LIN {X 0,Y 232.214,Z 369.64,A -85,B 0,C 180,E1 -19869.961,E2 -19869.961} C_VEL
LIN {X 0,Y 230.264,Z 376.571,A -85,B 0,C 180,E1 -19872.229,E2 -19872.229} C_VEL
LIN {X 0,Y 229.077,Z 381.074,A -85,B 0,C 180,E1 -19873.972,E2 -19873.972} C_VEL
LIN {X 0,Y 227.545,Z 386.565,A -85,B 0,C 180,E1 -19876.606,E2 -19876.606} C_VEL
LIN {X 0,Y 226.573,Z 390.894,A -85,B 0,C 180,E1 -19879.274,E2 -19879.274} C_VEL
LIN {X 0,Y 226.135,Z 393.264,A -85,B 0,C 180,E1 -19881.06,E2 -19881.06} C_VEL
LIN {X 0,Y 225.811,Z 395.066,A -85,B 0,C 180,E1 -19882.849,E2 -19882.849} C_VEL
LIN {X 0,Y 225.588,Z 397.52,A -85,B 0,C 180,E1 -19886.428,E2 -19886.428} C_VEL
LIN {X 0,Y 225.625,Z 398.113,A -85,B 0,C 180,E1 -19888.215,E2 -19888.215} C_VEL
LIN {X 0,Y 225.708,Z 398.27,A -85,B 0,C 180,E1 -19890,E2 -19890} C_VEL
LIN {X 0,Y 225.624,Z 398.113,A -85,B 0,C 180,E1 -19891.785,E2 -19891.785} C_VEL
LIN {X 0,Y 225.587,Z 397.046,A -85,B 0,C 180,E1 -19894.475,E2 -19894.475} C_VEL
LIN {X 0,Y 225.778,Z 395.065,A -85,B 0,C 180,E1 -19897.152,E2 -19897.152} C_VEL
LIN {X 0,Y 226.327,Z 392.112,A -85,B 0,C 180,E1 -19899.834,E2 -19899.834} C_VEL
LIN {X 0,Y 227.177,Z 388.12,A -85,B 0,C 180,E1 -19902.507,E2 -19902.507} C_VEL
LIN {X 0,Y 228.512,Z 382.989,A -85,B 0,C 180,E1 -19905.154,E2 -19905.154} C_VEL
LIN {X 0,Y 229.992,Z 377.728,A -85,B 0,C 180,E1 -19907.334,E2 -19907.334} C_VEL
LIN {X 0,Y 231.748,Z 371.413,A -85,B 0,C 180,E1 -19909.486,E2 -19909.486} C_VEL
LIN {X 0,Y 233.277,Z 365.461,A -85,B 0,C 180,E1 -19911.194,E2 -19911.194} C_VEL
LIN {X 0,Y 235.024,Z 358.534,A -85,B 0,C 180,E1 -19912.876,E2 -19912.876} C_VEL
LIN {X 0,Y 237.101,Z 350.359,A -85,B 0,C 180,E1 -19914.518,E2 -19914.518} C_VEL
LIN {X 0,Y 239.016,Z 341.85,A -85,B 0,C 180,E1 -19915.937,E2 -19915.937} C_VEL
LIN {X 0,Y 240.893,Z 333.14,A -85,B 0,C 180,E1 -19917.12,E2 -19917.12} C_VEL
LIN {X 0,Y 242.62,Z 323.384,A -85,B 0,C 180,E1 -19918.198,E2 -19918.198} C_VEL
LIN {X 0,Y 244.14,Z 313.306,A -85,B 0,C 180,E1 -19919.063,E2 -19919.063} C_VEL
LIN {X 0,Y 245.33,Z 303.86,A -85,B 0,C 180,E1 -19919.669,E2 -19919.669} C_VEL
LIN {X 0,Y 246.133,Z 293.823,A -85,B 0,C 180,E1 -19920.141,E2 -19920.141} C_VEL
LIN {X 0,Y 247.891,Z 250.011,A -85,B 0,C 180,E1 -19921.412,E2 -19921.412} C_VEL
LIN {X 0,Y 248.127,Z 242.633,A -85,B 0,C 180,E1 -19921.624,E2 -19921.624} C_VEL
LIN {X 0,Y 244.357,Z 220.685,A -85,B 0,C 180,E1 -19922.914,E2 -19922.914} C_VEL
LIN {X 0,Y 243.134,Z 215.724,A -85,B 0,C 180,E1 -19923.271,E2 -19923.271} C_VEL
LIN {X 0,Y 235.991,Z 199.45,A -85,B 0,C 180,E1 -19924.997,E2 -19924.997} C_VEL
LIN {X 0,Y 230.184,Z 187.454,A -85,B 0,C 180,E1 -19926.503,E2 -19926.503} C_VEL
LIN {X 0,Y 229.739,Z 185.681,A -85,B 0,C 180,E1 -19927.308,E2 -19927.308} C_VEL
LIN {X 0,Y 228.311,Z 179.722,A -85,B 0,C 180,E1 -19931.046,E2 -19931.046} C_VEL
LIN {X 0,Y 227.848,Z 177.605,A -85,B 0,C 180,E1 -19932.574,E2 -19932.574} C_VEL
LIN {X 0,Y 227.808,Z 177.611,A -85,B 0,C 180,E1 -19937.256,E2 -19937.256} C_VEL
LIN {X 0,Y 227.846,Z 177.6,A -85,B 0,C 180,E1 -19941.908,E2 -19941.908} C_VEL
LIN {X 0,Y 227.881,Z 177.572,A -85,B 0,C 180,E1 -19946.376,E2 -19946.376} C_VEL
LIN {X 0,Y 227.918,Z 177.586,A -85,B 0,C 180,E1 -19950.437,E2 -19950.437} C_VEL
LIN {X 0,Y 227.929,Z 177.566,A -85,B 0,C 180,E1 -19954.425,E2 -19954.425} C_VEL
LIN {X 0,Y 227.962,Z 177.578,A -85,B 0,C 180,E1 -19958.286,E2 -19958.286} C_VEL
LIN {X 0,Y 228.034,Z 177.546,A -85,B 0,C 180,E1 -19962.825,E2 -19962.825} C_VEL
LIN {X 0,Y 228.072,Z 177.558,A -85,B 0,C 180,E1 -19967.542,E2 -19967.542} C_VEL
LIN {X 0,Y 228.266,Z 177.506,A -85,B 0,C 180,E1 -19971.144,E2 -19971.144} C_VEL
LIN {X 0,Y 228.323,Z 177.524,A -85,B 0,C 180,E1 -19972.927,E2 -19972.927} C_VEL
LIN {X 0,Y 228.552,Z 177.483,A -85,B 0,C 180,E1 -19978.237,E2 -19978.237} C_VEL
LIN {X 0,Y 228.553,Z 177.478,A -85,B 0,C 180,E1 -19981.761,E2 -19981.761} C_VEL
LIN {X 0,Y 228.353,Z 177.524,A -85,B 0,C 180,E1 -19987.07,E2 -19987.07} C_VEL
LIN {X 0,Y 228.161,Z 177.521,A -85,B 0,C 180,E1 -19990.649,E2 -19990.649} C_VEL
LIN {X 0,Y 228.062,Z 177.578,A -85,B 0,C 180,E1 -19994.271,E2 -19994.271} C_VEL
LIN {X 0,Y 228,Z 177.547,A -85,B 0,C 180,E1 -19997.952,E2 -19997.952} C_VEL
LIN {X 0,Y 227.927,Z 177.588,A -85,B 0,C 180,E1 -20002.329,E2 -20002.329} C_VEL
LIN {X 0,Y 227.94,Z 177.56,A -85,B 0,C 180,E1 -20006.602,E2 -20006.602} C_VEL
LIN {X 0,Y 227.906,Z 177.594,A -85,B 0,C 180,E1 -20010.295,E2 -20010.295} C_VEL
LIN {X 0,Y 227.886,Z 177.573,A -85,B 0,C 180,E1 -20013.718,E2 -20013.718} C_VEL
LIN {X 0,Y 227.866,Z 177.602,A -85,B 0,C 180,E1 -20018.085,E2 -20018.085} C_VEL
LIN {X 0,Y 227.812,Z 177.605,A -85,B 0,C 180,E1 -20022.741,E2 -20022.741} C_VEL
LIN {X 0,Y 227.811,Z 177.543,A -85,B 0,C 180,E1 -20027.258,E2 -20027.258} C_VEL
LIN {X 0,Y 227.866,Z 177.603,A -85,B 0,C 180,E1 -20031.914,E2 -20031.914} C_VEL
LIN {X 0,Y 227.929,Z 177.929,A -85,B 0,C 180,E1 -20032.938,E2 -20032.938} C_VEL
LIN {X 0,Y 228.316,Z 179.228,A -85,B 0,C 180,E1 -20033.246,E2 -20033.246} C_VEL
LIN {X 0,Y 230.062,Z 181.874,A -85,B 0,C 180,E1 -20033.684,E2 -20033.684} C_VEL
LIN {X 0,Y 239.018,Z 197.391,A -85,B 0,C 180,E1 -20035.813,E2 -20035.813} C_VEL
LIN {X 0,Y 245.285,Z 209.395,A -85,B 0,C 180,E1 -20037.22,E2 -20037.22} C_VEL
LIN {X 0,Y 252.548,Z 222.93,A -85,B 0,C 180,E1 -20038.725,E2 -20038.725} C_VEL
LIN {X 0,Y 261.317,Z 235.879,A -85,B 0,C 180,E1 -20040.298,E2 -20040.298} C_VEL
LIN {X 0,Y 272.635,Z 249.159,A -85,B 0,C 180,E1 -20042.045,E2 -20042.045} C_VEL
LIN {X 0,Y 286.641,Z 263.214,A -85,B 0,C 180,E1 -20043.918,E2 -20043.918} C_VEL
LIN {X 0,Y 299.817,Z 274.419,A -85,B 0,C 180,E1 -20045.476,E2 -20045.476} C_VEL
LIN {X 0,Y 307.547,Z 280.739,A -85,B 0,C 180,E1 -20046.479,E2 -20046.479} C_VEL
LIN {X 0,Y 315.797,Z 287.099,A -85,B 0,C 180,E1 -20047.77,E2 -20047.77} C_VEL
LIN {X 0,Y 323.581,Z 292.925,A -85,B 0,C 180,E1 -20049.173,E2 -20049.173} C_VEL
LIN {X 0,Y 331.85,Z 299.062,A -85,B 0,C 180,E1 -20050.874,E2 -20050.874} C_VEL
LIN {X 0,Y 339.226,Z 304.074,A -85,B 0,C 180,E1 -20052.563,E2 -20052.563} C_VEL
LIN {X 0,Y 345.901,Z 309.055,A -85,B 0,C 180,E1 -20054.348,E2 -20054.348} C_VEL
LIN {X 0,Y 351.923,Z 312.847,A -85,B 0,C 180,E1 -20056.135,E2 -20056.135} C_VEL
LIN {X 0,Y 355.943,Z 315.097,A -85,B 0,C 180,E1 -20057.456,E2 -20057.456} C_VEL
LIN {X 0,Y 359.121,Z 317.594,A -85,B 0,C 180,E1 -20058.715,E2 -20058.715} C_VEL
LIN {X 0,Y 363.313,Z 320.464,A -85,B 0,C 180,E1 -20060.589,E2 -20060.589} C_VEL
LIN {X 0,Y 366.561,Z 322.302,A -85,B 0,C 180,E1 -20062.287,E2 -20062.287} C_VEL
LIN {X 0,Y 368.408,Z 323.209,A -85,B 0,C 180,E1 -20063.428,E2 -20063.428} C_VEL
LIN {X 0,Y 369.964,Z 323.883,A -85,B 0,C 180,E1 -20064.55,E2 -20064.55} C_VEL
LIN {X 0,Y 371.235,Z 324.349,A -85,B 0,C 180,E1 -20065.657,E2 -20065.657} C_VEL
LIN {X 0,Y 372.231,Z 324.627,A -85,B 0,C 180,E1 -20066.753,E2 -20066.753} C_VEL
LIN {X 0,Y 372.866,Z 324.996,A -85,B 0,C 180,E1 -20067.84,E2 -20067.84} C_VEL
LIN {X 0,Y 373.221,Z 325.279,A -85,B 0,C 180,E1 -20068.921,E2 -20068.921} C_VEL
LIN {X 0,Y 373.406,Z 325.182,A -85,B 0,C 180,E1 -20070,E2 -20070} C_VEL
LIN {X 0,Y 373.242,Z 325.214,A -85,B 0,C 180,E1 -20071.079,E2 -20071.079} C_VEL
LIN {X 0,Y 372.792,Z 324.929,A -85,B 0,C 180,E1 -20072.349,E2 -20072.349} C_VEL
LIN {X 0,Y 371.247,Z 324.325,A -85,B 0,C 180,E1 -20074.343,E2 -20074.343} C_VEL
LIN {X 0,Y 369.974,Z 323.88,A -85,B 0,C 180,E1 -20075.45,E2 -20075.45} C_VEL
LIN {X 0,Y 368.057,Z 323.044,A -85,B 0,C 180,E1 -20076.821,E2 -20076.821} C_VEL
LIN {X 0,Y 366.574,Z 322.333,A -85,B 0,C 180,E1 -20077.713,E2 -20077.713} C_VEL
LIN {X 0,Y 363.308,Z 320.439,A -85,B 0,C 180,E1 -20079.406,E2 -20079.406} C_VEL
LIN {X 0,Y 359.112,Z 317.577,A -85,B 0,C 180,E1 -20081.286,E2 -20081.286} C_VEL
LIN {X 0,Y 355.896,Z 315.079,A -85,B 0,C 180,E1 -20082.546,E2 -20082.546} C_VEL
LIN {X 0,Y 351.917,Z 312.837,A -85,B 0,C 180,E1 -20083.866,E2 -20083.866} C_VEL
LIN {X 0,Y 345.745,Z 308.908,A -85,B 0,C 180,E1 -20085.699,E2 -20085.699} C_VEL
LIN {X 0,Y 338.798,Z 303.827,A -85,B 0,C 180,E1 -20087.534,E2 -20087.534} C_VEL
LIN {X 0,Y 330.886,Z 298.432,A -85,B 0,C 180,E1 -20089.33,E2 -20089.33} C_VEL
LIN {X 0,Y 323.177,Z 292.616,A -85,B 0,C 180,E1 -20090.901,E2 -20090.901} C_VEL
LIN {X 0,Y 315.363,Z 286.776,A -85,B 0,C 180,E1 -20092.3,E2 -20092.3} C_VEL
LIN {X 0,Y 306.83,Z 280.18,A -85,B 0,C 180,E1 -20093.624,E2 -20093.624} C_VEL
LIN {X 0,Y 298.134,Z 273.077,A -85,B 0,C 180,E1 -20094.73,E2 -20094.73} C_VEL
LIN {X 0,Y 282.857,Z 259.613,A -85,B 0,C 180,E1 -20096.561,E2 -20096.561} C_VEL
LIN {X 0,Y 269.247,Z 245.479,A -85,B 0,C 180,E1 -20098.451,E2 -20098.451} C_VEL
LIN {X 0,Y 260.422,Z 234.592,A -85,B 0,C 180,E1 -20099.856,E2 -20099.856} C_VEL
LIN {X 0,Y 252.398,Z 222.675,A -85,B 0,C 180,E1 -20101.304,E2 -20101.304} C_VEL
LIN {X 0,Y 245.458,Z 209.83,A -85,B 0,C 180,E1 -20102.739,E2 -20102.739} C_VEL
LIN {X 0,Y 239.261,Z 197.815,A -85,B 0,C 180,E1 -20104.132,E2 -20104.132} C_VEL
LIN {X 0,Y 231.588,Z 184.592,A -85,B 0,C 180,E1 -20105.935,E2 -20105.935} C_VEL
LIN {X 0,Y 229.701,Z 181.488,A -85,B 0,C 180,E1 -20106.397,E2 -20106.397} C_VEL
LIN {X 0,Y 228.091,Z 178.529,A -85,B 0,C 180,E1 -20106.86,E2 -20106.86} C_VEL
LIN {X 0,Y 227.9,Z 177.655,A -85,B 0,C 180,E1 -20107.312,E2 -20107.312} C_VEL
LIN {X 0,Y 227.829,Z 177.552,A -85,B 0,C 180,E1 -20110.375,E2 -20110.375} C_VEL
LIN {X 0,Y 227.832,Z 177.581,A -85,B 0,C 180,E1 -20115.193,E2 -20115.193} C_VEL
LIN {X 0,Y 227.83,Z 177.584,A -85,B 0,C 180,E1 -20119.625,E2 -20119.625} C_VEL
LIN {X 0,Y 227.896,Z 177.578,A -85,B 0,C 180,E1 -20124.132,E2 -20124.132} C_VEL
LIN {X 0,Y 227.87,Z 177.6,A -85,B 0,C 180,E1 -20128.379,E2 -20128.379} C_VEL
LIN {X 0,Y 227.883,Z 177.565,A -85,B 0,C 180,E1 -20132.446,E2 -20132.446} C_VEL
LIN {X 0,Y 227.911,Z 177.596,A -85,B 0,C 180,E1 -20136.368,E2 -20136.368} C_VEL
LIN {X 0,Y 227.939,Z 177.552,A -85,B 0,C 180,E1 -20140.175,E2 -20140.175} C_VEL
LIN {X 0,Y 228.055,Z 177.569,A -85,B 0,C 180,E1 -20143.899,E2 -20143.899} C_VEL
LIN {X 0,Y 228.092,Z 177.554,A -85,B 0,C 180,E1 -20147.545,E2 -20147.545} C_VEL
LIN {X 0,Y 228.304,Z 177.505,A -85,B 0,C 180,E1 -20151.147,E2 -20151.147} C_VEL
LIN {X 0,Y 228.353,Z 177.524,A -85,B 0,C 180,E1 -20152.93,E2 -20152.93} C_VEL
LIN {X 0,Y 228.553,Z 177.478,A -85,B 0,C 180,E1 -20158.239,E2 -20158.239} C_VEL
LIN {X 0,Y 228.552,Z 177.483,A -85,B 0,C 180,E1 -20161.763,E2 -20161.763} C_VEL
LIN {X 0,Y 228.323,Z 177.524,A -85,B 0,C 180,E1 -20167.073,E2 -20167.073} C_VEL
LIN {X 0,Y 228.145,Z 177.523,A -85,B 0,C 180,E1 -20170.652,E2 -20170.652} C_VEL
LIN {X 0,Y 228.064,Z 177.573,A -85,B 0,C 180,E1 -20174.273,E2 -20174.273} C_VEL
LIN {X 0,Y 228.003,Z 177.542,A -85,B 0,C 180,E1 -20177.954,E2 -20177.954} C_VEL
LIN {X 0,Y 227.93,Z 177.589,A -85,B 0,C 180,E1 -20182.33,E2 -20182.33} C_VEL
LIN {X 0,Y 227.943,Z 177.556,A -85,B 0,C 180,E1 -20186.604,E2 -20186.604} C_VEL
LIN {X 0,Y 227.908,Z 177.595,A -85,B 0,C 180,E1 -20190.297,E2 -20190.297} C_VEL
LIN {X 0,Y 227.879,Z 177.572,A -85,B 0,C 180,E1 -20193.721,E2 -20193.721} C_VEL
LIN {X 0,Y 227.846,Z 177.6,A -85,B 0,C 180,E1 -20198.092,E2 -20198.092} C_VEL
LIN {X 0,Y 227.808,Z 177.609,A -85,B 0,C 180,E1 -20202.744,E2 -20202.744} C_VEL
LIN {X 0,Y 227.85,Z 177.623,A -85,B 0,C 180,E1 -20207.506,E2 -20207.506} C_VEL
LIN {X 0,Y 229.254,Z 183.3,A -85,B 0,C 180,E1 -20211.23,E2 -20211.23} C_VEL
LIN {X 0,Y 230.082,Z 187.069,A -85,B 0,C 180,E1 -20213.403,E2 -20213.403} C_VEL
LIN {X 0,Y 231.752,Z 190.832,A -85,B 0,C 180,E1 -20213.949,E2 -20213.949} C_VEL
LIN {X 0,Y 238.601,Z 205.182,A -85,B 0,C 180,E1 -20215.643,E2 -20215.643} C_VEL
LIN {X 0,Y 243.547,Z 216.733,A -85,B 0,C 180,E1 -20216.827,E2 -20216.827} C_VEL
LIN {X 0,Y 247.169,Z 236.517,A -85,B 0,C 180,E1 -20218.035,E2 -20218.035} C_VEL
LIN {X 0,Y 248.164,Z 243.57,A -85,B 0,C 180,E1 -20218.412,E2 -20218.412} C_VEL
LIN {X 0,Y 248.06,Z 246.228,A -85,B 0,C 180,E1 -20218.486,E2 -20218.486} C_VEL
LIN {X 0,Y 247.255,Z 252.073,A -85,B 0,C 180,E1 -20218.567,E2 -20218.567} C_VEL
LIN {X 0,Y 241.602,Z 271.074,A -85,B 0,C 180,E1 -20218.4,E2 -20218.4} C_VEL
LIN {X 0,Y 240.823,Z 276.917,A -85,B 0,C 180,E1 -20218.487,E2 -20218.487} C_VEL
LIN {X 0,Y 239.896,Z 296.606,A -85,B 0,C 180,E1 -20219.126,E2 -20219.126} C_VEL
LIN {X 0,Y 238.338,Z 310.54,A -85,B 0,C 180,E1 -20219.915,E2 -20219.915} C_VEL
LIN {X 0,Y 236.759,Z 321.18,A -85,B 0,C 180,E1 -20220.795,E2 -20220.795} C_VEL
LIN {X 0,Y 235.242,Z 329.685,A -85,B 0,C 180,E1 -20221.688,E2 -20221.688} C_VEL
LIN {X 0,Y 233.324,Z 338.958,A -85,B 0,C 180,E1 -20222.898,E2 -20222.898} C_VEL
LIN {X 0,Y 231.165,Z 347.897,A -85,B 0,C 180,E1 -20224.327,E2 -20224.327} C_VEL
LIN {X 0,Y 228.986,Z 356.423,A -85,B 0,C 180,E1 -20226.005,E2 -20226.005} C_VEL
LIN {X 0,Y 227.032,Z 363.64,A -85,B 0,C 180,E1 -20227.715,E2 -20227.715} C_VEL
LIN {X 0,Y 225.349,Z 370.062,A -85,B 0,C 180,E1 -20229.536,E2 -20229.536} C_VEL
LIN {X 0,Y 223.482,Z 376.379,A -85,B 0,C 180,E1 -20231.671,E2 -20231.671} C_VEL
LIN {X 0,Y 222.246,Z 380.882,A -85,B 0,C 180,E1 -20233.465,E2 -20233.465} C_VEL
LIN {X 0,Y 220.607,Z 386.372,A -85,B 0,C 180,E1 -20236.177,E2 -20236.177} C_VEL
LIN {X 0,Y 219.584,Z 390.702,A -85,B 0,C 180,E1 -20238.929,E2 -20238.929} C_VEL
LIN {X 0,Y 219.086,Z 393.072,A -85,B 0,C 180,E1 -20240.77,E2 -20240.77} C_VEL
LIN {X 0,Y 218.737,Z 394.874,A -85,B 0,C 180,E1 -20242.616,E2 -20242.616} C_VEL
LIN {X 0,Y 218.501,Z 397.328,A -85,B 0,C 180,E1 -20246.312,E2 -20246.312} C_VEL
LIN {X 0,Y 218.525,Z 397.921,A -85,B 0,C 180,E1 -20248.157,E2 -20248.157} C_VEL
LIN {X 0,Y 218.623,Z 398.079,A -85,B 0,C 180,E1 -20250,E2 -20250} C_VEL
LIN {X 0,Y 218.524,Z 397.921,A -85,B 0,C 180,E1 -20251.843,E2 -20251.843} C_VEL
LIN {X 0,Y 218.484,Z 397.064,A -85,B 0,C 180,E1 -20254.292,E2 -20254.292} C_VEL
LIN {X 0,Y 218.705,Z 394.873,A -85,B 0,C 180,E1 -20257.385,E2 -20257.385} C_VEL
LIN {X 0,Y 219.313,Z 391.92,A -85,B 0,C 180,E1 -20260.151,E2 -20260.151} C_VEL
LIN {X 0,Y 220.202,Z 387.927,A -85,B 0,C 180,E1 -20262.909,E2 -20262.909} C_VEL
LIN {X 0,Y 221.652,Z 382.797,A -85,B 0,C 180,E1 -20265.635,E2 -20265.635} C_VEL
LIN {X 0,Y 223.161,Z 377.535,A -85,B 0,C 180,E1 -20267.882,E2 -20267.882} C_VEL
LIN {X 0,Y 225.05,Z 371.221,A -85,B 0,C 180,E1 -20270.091,E2 -20270.091} C_VEL
LIN {X 0,Y 226.622,Z 365.268,A -85,B 0,C 180,E1 -20271.848,E2 -20271.848} C_VEL
LIN {X 0,Y 228.474,Z 358.341,A -85,B 0,C 180,E1 -20273.571,E2 -20273.571} C_VEL
LIN {X 0,Y 230.662,Z 350.168,A -85,B 0,C 180,E1 -20275.249,E2 -20275.249} C_VEL
LIN {X 0,Y 232.638,Z 341.658,A -85,B 0,C 180,E1 -20276.703,E2 -20276.703} C_VEL
LIN {X 0,Y 234.602,Z 332.948,A -85,B 0,C 180,E1 -20277.909,E2 -20277.909} C_VEL
LIN {X 0,Y 236.379,Z 323.192,A -85,B 0,C 180,E1 -20279.012,E2 -20279.012} C_VEL
LIN {X 0,Y 237.942,Z 313.114,A -85,B 0,C 180,E1 -20279.896,E2 -20279.896} C_VEL
LIN {X 0,Y 239.227,Z 303.118,A -85,B 0,C 180,E1 -20280.544,E2 -20280.544} C_VEL
LIN {X 0,Y 240.04,Z 293.142,A -85,B 0,C 180,E1 -20281.012,E2 -20281.012} C_VEL
LIN {X 0,Y 242.113,Z 243.843,A -85,B 0,C 180,E1 -20282.457,E2 -20282.457} C_VEL
LIN {X 0,Y 238.247,Z 221.322,A -85,B 0,C 180,E1 -20283.841,E2 -20283.841} C_VEL
LIN {X 0,Y 237.362,Z 218.29,A -85,B 0,C 180,E1 -20284.091,E2 -20284.091} C_VEL
LIN {X 0,Y 230.872,Z 203.304,A -85,B 0,C 180,E1 -20285.74,E2 -20285.74} C_VEL
LIN {X 0,Y 224.409,Z 190.406,A -85,B 0,C 180,E1 -20287.434,E2 -20287.434} C_VEL
LIN {X 0,Y 222.782,Z 186.821,A -85,B 0,C 180,E1 -20288.007,E2 -20288.007} C_VEL
LIN {X 0,Y 221.299,Z 180.788,A -85,B 0,C 180,E1 -20291.829,E2 -20291.829} C_VEL
LIN {X 0,Y 220.782,Z 178.503,A -85,B 0,C 180,E1 -20293.481,E2 -20293.481} C_VEL
LIN {X 0,Y 220.768,Z 178.482,A -85,B 0,C 180,E1 -20298.046,E2 -20298.046} C_VEL
LIN {X 0,Y 220.825,Z 178.479,A -85,B 0,C 180,E1 -20302.792,E2 -20302.792} C_VEL
LIN {X 0,Y 220.819,Z 178.459,A -85,B 0,C 180,E1 -20307.243,E2 -20307.243} C_VEL
LIN {X 0,Y 220.836,Z 178.451,A -85,B 0,C 180,E1 -20311.485,E2 -20311.485} C_VEL
LIN {X 0,Y 220.868,Z 178.46,A -85,B 0,C 180,E1 -20315.564,E2 -20315.564} C_VEL
LIN {X 0,Y 220.892,Z 178.438,A -85,B 0,C 180,E1 -20319.513,E2 -20319.513} C_VEL
LIN {X 0,Y 221.016,Z 178.427,A -85,B 0,C 180,E1 -20323.369,E2 -20323.369} C_VEL
LIN {X 0,Y 221.011,Z 178.444,A -85,B 0,C 180,E1 -20327.138,E2 -20327.138} C_VEL
LIN {X 0,Y 221.204,Z 178.383,A -85,B 0,C 180,E1 -20330.858,E2 -20330.858} C_VEL
LIN {X 0,Y 221.258,Z 178.398,A -85,B 0,C 180,E1 -20332.7,E2 -20332.7} C_VEL
LIN {X 0,Y 221.51,Z 178.36,A -85,B 0,C 180,E1 -20338.181,E2 -20338.181} C_VEL
LIN {X 0,Y 221.511,Z 178.355,A -85,B 0,C 180,E1 -20341.817,E2 -20341.817} C_VEL
LIN {X 0,Y 221.288,Z 178.399,A -85,B 0,C 180,E1 -20347.297,E2 -20347.297} C_VEL
LIN {X 0,Y 221.11,Z 178.401,A -85,B 0,C 180,E1 -20350.993,E2 -20350.993} C_VEL
LIN {X 0,Y 221.014,Z 178.436,A -85,B 0,C 180,E1 -20356.629,E2 -20356.629} C_VEL
LIN {X 0,Y 220.89,Z 178.436,A -85,B 0,C 180,E1 -20360.485,E2 -20360.485} C_VEL
LIN {X 0,Y 220.865,Z 178.469,A -85,B 0,C 180,E1 -20364.434,E2 -20364.434} C_VEL
LIN {X 0,Y 220.833,Z 178.449,A -85,B 0,C 180,E1 -20368.513,E2 -20368.513} C_VEL
LIN {X 0,Y 220.821,Z 178.463,A -85,B 0,C 180,E1 -20372.754,E2 -20372.754} C_VEL
LIN {X 0,Y 220.835,Z 178.477,A -85,B 0,C 180,E1 -20377.287,E2 -20377.287} C_VEL
LIN {X 0,Y 220.772,Z 178.47,A -85,B 0,C 180,E1 -20381.951,E2 -20381.951} C_VEL
LIN {X 0,Y 220.772,Z 178.441,A -85,B 0,C 180,E1 -20385.546,E2 -20385.546} C_VEL
LIN {X 0,Y 220.805,Z 178.44,A -85,B 0,C 180,E1 -20390.463,E2 -20390.463} C_VEL
LIN {X 0,Y 220.869,Z 178.776,A -85,B 0,C 180,E1 -20391.555,E2 -20391.555} C_VEL
LIN {X 0,Y 221.231,Z 180.131,A -85,B 0,C 180,E1 -20391.89,E2 -20391.89} C_VEL
LIN {X 0,Y 222.982,Z 182.764,A -85,B 0,C 180,E1 -20392.361,E2 -20392.361} C_VEL
LIN {X 0,Y 230.22,Z 194.713,A -85,B 0,C 180,E1 -20394.2,E2 -20394.2} C_VEL
LIN {X 0,Y 238.43,Z 209.905,A -85,B 0,C 180,E1 -20396.163,E2 -20396.163} C_VEL
LIN {X 0,Y 246.332,Z 225.31,A -85,B 0,C 180,E1 -20397.917,E2 -20397.917} C_VEL
LIN {X 0,Y 254.125,Z 237.265,A -85,B 0,C 180,E1 -20399.406,E2 -20399.406} C_VEL
LIN {X 0,Y 261.098,Z 246.325,A -85,B 0,C 180,E1 -20400.594,E2 -20400.594} C_VEL
LIN {X 0,Y 272.34,Z 258.902,A -85,B 0,C 180,E1 -20402.297,E2 -20402.297} C_VEL
LIN {X 0,Y 285.178,Z 271.16,A -85,B 0,C 180,E1 -20403.991,E2 -20403.991} C_VEL
LIN {X 0,Y 298.365,Z 282.288,A -85,B 0,C 180,E1 -20405.579,E2 -20405.579} C_VEL
LIN {X 0,Y 306.925,Z 289.092,A -85,B 0,C 180,E1 -20406.771,E2 -20406.771} C_VEL
LIN {X 0,Y 315.592,Z 295.809,A -85,B 0,C 180,E1 -20408.207,E2 -20408.207} C_VEL
LIN {X 0,Y 323.961,Z 301.874,A -85,B 0,C 180,E1 -20409.783,E2 -20409.783} C_VEL
LIN {X 0,Y 331.81,Z 307.611,A -85,B 0,C 180,E1 -20411.476,E2 -20411.476} C_VEL
LIN {X 0,Y 338.558,Z 312.236,A -85,B 0,C 180,E1 -20413.105,E2 -20413.105} C_VEL
LIN {X 0,Y 343.959,Z 316.177,A -85,B 0,C 180,E1 -20414.596,E2 -20414.596} C_VEL
LIN {X 0,Y 348.699,Z 319.119,A -85,B 0,C 180,E1 -20416.004,E2 -20416.004} C_VEL
LIN {X 0,Y 352.904,Z 321.471,A -85,B 0,C 180,E1 -20417.372,E2 -20417.372} C_VEL
LIN {X 0,Y 357.621,Z 325.06,A -85,B 0,C 180,E1 -20419.293,E2 -20419.293} C_VEL
LIN {X 0,Y 361.369,Z 327.489,A -85,B 0,C 180,E1 -20421.049,E2 -20421.049} C_VEL
LIN {X 0,Y 363.545,Z 328.713,A -85,B 0,C 180,E1 -20422.223,E2 -20422.223} C_VEL
LIN {X 0,Y 365.441,Z 329.628,A -85,B 0,C 180,E1 -20423.374,E2 -20423.374} C_VEL
LIN {X 0,Y 367.1,Z 330.364,A -85,B 0,C 180,E1 -20424.568,E2 -20424.568} C_VEL
LIN {X 0,Y 368.306,Z 330.811,A -85,B 0,C 180,E1 -20425.623,E2 -20425.623} C_VEL
LIN {X 0,Y 369.322,Z 331.105,A -85,B 0,C 180,E1 -20426.727,E2 -20426.727} C_VEL
LIN {X 0,Y 369.972,Z 331.455,A -85,B 0,C 180,E1 -20427.823,E2 -20427.823} C_VEL
LIN {X 0,Y 370.325,Z 331.734,A -85,B 0,C 180,E1 -20428.913,E2 -20428.913} C_VEL
LIN {X 0,Y 370.523,Z 331.644,A -85,B 0,C 180,E1 -20430,E2 -20430} C_VEL
LIN {X 0,Y 370.339,Z 331.689,A -85,B 0,C 180,E1 -20431.087,E2 -20431.087} C_VEL
LIN {X 0,Y 369.977,Z 331.421,A -85,B 0,C 180,E1 -20432.177,E2 -20432.177} C_VEL
LIN {X 0,Y 369.32,Z 331.082,A -85,B 0,C 180,E1 -20433.273,E2 -20433.273} C_VEL
LIN {X 0,Y 368.309,Z 330.779,A -85,B 0,C 180,E1 -20434.377,E2 -20434.377} C_VEL
LIN {X 0,Y 367.016,Z 330.323,A -85,B 0,C 180,E1 -20435.494,E2 -20435.494} C_VEL
LIN {X 0,Y 365.437,Z 329.642,A -85,B 0,C 180,E1 -20436.626,E2 -20436.626} C_VEL
LIN {X 0,Y 362.342,Z 328.045,A -85,B 0,C 180,E1 -20438.435,E2 -20438.435} C_VEL
LIN {X 0,Y 358.864,Z 325.916,A -85,B 0,C 180,E1 -20440.152,E2 -20440.152} C_VEL
LIN {X 0,Y 354.955,Z 323.141,A -85,B 0,C 180,E1 -20441.812,E2 -20441.812} C_VEL
LIN {X 0,Y 352.801,Z 321.444,A -85,B 0,C 180,E1 -20442.658,E2 -20442.658} C_VEL
LIN {X 0,Y 347.992,Z 318.709,A -85,B 0,C 180,E1 -20444.213,E2 -20444.213} C_VEL
LIN {X 0,Y 343.044,Z 315.551,A -85,B 0,C 180,E1 -20445.66,E2 -20445.66} C_VEL
LIN {X 0,Y 338.086,Z 311.947,A -85,B 0,C 180,E1 -20447.017,E2 -20447.017} C_VEL
LIN {X 0,Y 330.772,Z 306.921,A -85,B 0,C 180,E1 -20448.753,E2 -20448.753} C_VEL
LIN {X 0,Y 323.263,Z 301.326,A -85,B 0,C 180,E1 -20450.356,E2 -20450.356} C_VEL
LIN {X 0,Y 314.609,Z 295.066,A -85,B 0,C 180,E1 -20451.969,E2 -20451.969} C_VEL
LIN {X 0,Y 306.168,Z 288.54,A -85,B 0,C 180,E1 -20453.34,E2 -20453.34} C_VEL
LIN {X 0,Y 298.371,Z 282.29,A -85,B 0,C 180,E1 -20454.423,E2 -20454.423} C_VEL
LIN {X 0,Y 286.498,Z 272.292,A -85,B 0,C 180,E1 -20455.848,E2 -20455.848} C_VEL
LIN {X 0,Y 276.553,Z 263.037,A -85,B 0,C 180,E1 -20457.124,E2 -20457.124} C_VEL
LIN {X 0,Y 264.555,Z 250.461,A -85,B 0,C 180,E1 -20458.856,E2 -20458.856} C_VEL
LIN {X 0,Y 255.684,Z 239.447,A -85,B 0,C 180,E1 -20460.317,E2 -20460.317} C_VEL
LIN {X 0,Y 247.844,Z 227.763,A -85,B 0,C 180,E1 -20461.781,E2 -20461.781} C_VEL
LIN {X 0,Y 241.06,Z 215.332,A -85,B 0,C 180,E1 -20463.226,E2 -20463.226} C_VEL
LIN {X 0,Y 234.477,Z 202.332,A -85,B 0,C 180,E1 -20464.769,E2 -20464.769} C_VEL
LIN {X 0,Y 225.477,Z 186.693,A -85,B 0,C 180,E1 -20466.994,E2 -20466.994} C_VEL
LIN {X 0,Y 222.661,Z 182.415,A -85,B 0,C 180,E1 -20467.717,E2 -20467.717} C_VEL
LIN {X 0,Y 221.064,Z 179.607,A -85,B 0,C 180,E1 -20468.186,E2 -20468.186} C_VEL
LIN {X 0,Y 220.856,Z 178.685,A -85,B 0,C 180,E1 -20468.516,E2 -20468.516} C_VEL
LIN {X 0,Y 220.771,Z 178.417,A -85,B 0,C 180,E1 -20471.952,E2 -20471.952} C_VEL
LIN {X 0,Y 220.772,Z 178.467,A -85,B 0,C 180,E1 -20475.547,E2 -20475.547} C_VEL
LIN {X 0,Y 220.806,Z 178.464,A -85,B 0,C 180,E1 -20480.464,E2 -20480.464} C_VEL
LIN {X 0,Y 220.829,Z 178.478,A -85,B 0,C 180,E1 -20482.795,E2 -20482.795} C_VEL
LIN {X 0,Y 220.821,Z 178.463,A -85,B 0,C 180,E1 -20487.246,E2 -20487.246} C_VEL
LIN {X 0,Y 220.833,Z 178.449,A -85,B 0,C 180,E1 -20491.487,E2 -20491.487} C_VEL
LIN {X 0,Y 220.865,Z 178.469,A -85,B 0,C 180,E1 -20495.566,E2 -20495.566} C_VEL
LIN {X 0,Y 220.89,Z 178.436,A -85,B 0,C 180,E1 -20499.515,E2 -20499.515} C_VEL
LIN {X 0,Y 221.014,Z 178.436,A -85,B 0,C 180,E1 -20503.371,E2 -20503.371} C_VEL
LIN {X 0,Y 221.11,Z 178.401,A -85,B 0,C 180,E1 -20509.007,E2 -20509.007} C_VEL
LIN {X 0,Y 221.288,Z 178.399,A -85,B 0,C 180,E1 -20512.703,E2 -20512.703} C_VEL
LIN {X 0,Y 221.511,Z 178.355,A -85,B 0,C 180,E1 -20518.183,E2 -20518.183} C_VEL
LIN {X 0,Y 221.51,Z 178.36,A -85,B 0,C 180,E1 -20521.819,E2 -20521.819} C_VEL
LIN {X 0,Y 221.258,Z 178.398,A -85,B 0,C 180,E1 -20527.3,E2 -20527.3} C_VEL
LIN {X 0,Y 221.067,Z 178.407,A -85,B 0,C 180,E1 -20530.997,E2 -20530.997} C_VEL
LIN {X 0,Y 220.996,Z 178.454,A -85,B 0,C 180,E1 -20534.74,E2 -20534.74} C_VEL
LIN {X 0,Y 220.922,Z 178.421,A -85,B 0,C 180,E1 -20538.55,E2 -20538.55} C_VEL
LIN {X 0,Y 220.896,Z 178.466,A -85,B 0,C 180,E1 -20542.684,E2 -20542.684} C_VEL
LIN {X 0,Y 220.886,Z 178.434,A -85,B 0,C 180,E1 -20547.016,E2 -20547.016} C_VEL
LIN {X 0,Y 220.864,Z 178.475,A -85,B 0,C 180,E1 -20550.779,E2 -20550.779} C_VEL
LIN {X 0,Y 220.803,Z 178.455,A -85,B 0,C 180,E1 -20554.956,E2 -20554.956} C_VEL
LIN {X 0,Y 220.807,Z 178.462,A -85,B 0,C 180,E1 -20559.538,E2 -20559.538} C_VEL
LIN {X 0,Y 220.771,Z 178.472,A -85,B 0,C 180,E1 -20564.456,E2 -20564.456} C_VEL
LIN {X 0,Y 220.775,Z 178.598,A -85,B 0,C 180,E1 -20566.647,E2 -20566.647} C_VEL
LIN {X 0,Y 222.587,Z 185.992,A -85,B 0,C 180,E1 -20571.583,E2 -20571.583} C_VEL
LIN {X 0,Y 222.872,Z 187.212,A -85,B 0,C 180,E1 -20572.094,E2 -20572.094} C_VEL
LIN {X 0,Y 229.383,Z 200.201,A -85,B 0,C 180,E1 -20573.876,E2 -20573.876} C_VEL
LIN {X 0,Y 236.388,Z 215.903,A -85,B 0,C 180,E1 -20575.664,E2 -20575.664} C_VEL
LIN {X 0,Y 238.114,Z 220.604,A -85,B 0,C 180,E1 -20576.112,E2 -20576.112} C_VEL
LIN {X 0,Y 241.471,Z 239.821,A -85,B 0,C 180,E1 -20577.308,E2 -20577.308} C_VEL
LIN {X 0,Y 242.105,Z 244.219,A -85,B 0,C 180,E1 -20577.555,E2 -20577.555} C_VEL
LIN {X 0,Y 240.823,Z 276.917,A -85,B 0,C 180,E1 -20578.487,E2 -20578.487} C_VEL
LIN {X 0,Y 240.034,Z 282.764,A -85,B 0,C 180,E1 -20578.572,E2 -20578.572} C_VEL
LIN {X 0,Y 237.099,Z 292.244,A -85,B 0,C 180,E1 -20578.517,E2 -20578.517} C_VEL
LIN {X 0,Y 233.891,Z 301.632,A -85,B 0,C 180,E1 -20578.575,E2 -20578.575} C_VEL
LIN {X 0,Y 232.666,Z 307.332,A -85,B 0,C 180,E1 -20578.822,E2 -20578.822} C_VEL
LIN {X 0,Y 230.755,Z 319.981,A -85,B 0,C 180,E1 -20579.833,E2 -20579.833} C_VEL
LIN {X 0,Y 228.985,Z 329.493,A -85,B 0,C 180,E1 -20580.841,E2 -20580.841} C_VEL
LIN {X 0,Y 227.018,Z 338.766,A -85,B 0,C 180,E1 -20582.08,E2 -20582.08} C_VEL
LIN {X 0,Y 224.774,Z 347.705,A -85,B 0,C 180,E1 -20583.542,E2 -20583.542} C_VEL
LIN {X 0,Y 222.492,Z 356.231,A -85,B 0,C 180,E1 -20585.258,E2 -20585.258} C_VEL
LIN {X 0,Y 220.445,Z 363.447,A -85,B 0,C 180,E1 -20587.012,E2 -20587.012} C_VEL
LIN {X 0,Y 218.737,Z 369.381,A -85,B 0,C 180,E1 -20588.714,E2 -20588.714} C_VEL
LIN {X 0,Y 216.734,Z 376.187,A -85,B 0,C 180,E1 -20591.079,E2 -20591.079} C_VEL
LIN {X 0,Y 215.438,Z 380.69,A -85,B 0,C 180,E1 -20592.927,E2 -20592.927} C_VEL
LIN {X 0,Y 213.693,Z 386.18,A -85,B 0,C 180,E1 -20595.72,E2 -20595.72} C_VEL
LIN {X 0,Y 212.571,Z 390.509,A -85,B 0,C 180,E1 -20598.558,E2 -20598.558} C_VEL
LIN {X 0,Y 212.06,Z 392.879,A -85,B 0,C 180,E1 -20600.462,E2 -20600.462} C_VEL
LIN {X 0,Y 211.493,Z 396.074,A -85,B 0,C 180,E1 -20604.279,E2 -20604.279} C_VEL
LIN {X 0,Y 211.42,Z 397.136,A -85,B 0,C 180,E1 -20606.188,E2 -20606.188} C_VEL
LIN {X 0,Y 211.427,Z 397.729,A -85,B 0,C 180,E1 -20608.095,E2 -20608.095} C_VEL
LIN {X 0,Y 211.539,Z 397.888,A -85,B 0,C 180,E1 -20610,E2 -20610} C_VEL
LIN {X 0,Y 211.426,Z 397.729,A -85,B 0,C 180,E1 -20611.905,E2 -20611.905} C_VEL
LIN {X 0,Y 211.396,Z 397.02,A -85,B 0,C 180,E1 -20614.145,E2 -20614.145} C_VEL
LIN {X 0,Y 211.646,Z 394.68,A -85,B 0,C 180,E1 -20617.633,E2 -20617.633} C_VEL
LIN {X 0,Y 212.3,Z 391.727,A -85,B 0,C 180,E1 -20620.49,E2 -20620.49} C_VEL
LIN {X 0,Y 213.241,Z 387.734,A -85,B 0,C 180,E1 -20623.338,E2 -20623.338} C_VEL
LIN {X 0,Y 214.784,Z 382.604,A -85,B 0,C 180,E1 -20626.148,E2 -20626.148} C_VEL
LIN {X 0,Y 216.367,Z 377.342,A -85,B 0,C 180,E1 -20628.463,E2 -20628.463} C_VEL
LIN {X 0,Y 218.364,Z 371.028,A -85,B 0,C 180,E1 -20630.734,E2 -20630.734} C_VEL
LIN {X 0,Y 220.012,Z 365.075,A -85,B 0,C 180,E1 -20632.54,E2 -20632.54} C_VEL
LIN {X 0,Y 221.981,Z 358.15,A -85,B 0,C 180,E1 -20634.304,E2 -20634.304} C_VEL
LIN {X 0,Y 224.244,Z 349.975,A -85,B 0,C 180,E1 -20636.025,E2 -20636.025} C_VEL
LIN {X 0,Y 226.317,Z 341.466,A -85,B 0,C 180,E1 -20637.511,E2 -20637.511} C_VEL
LIN {X 0,Y 228.352,Z 332.757,A -85,B 0,C 180,E1 -20638.743,E2 -20638.743} C_VEL
LIN {X 0,Y 230.194,Z 323.001,A -85,B 0,C 180,E1 -20639.87,E2 -20639.87} C_VEL
LIN {X 0,Y 231.635,Z 314.21,A -85,B 0,C 180,E1 -20640.671,E2 -20640.671} C_VEL
LIN {X 0,Y 233.049,Z 303.89,A -85,B 0,C 180,E1 -20641.374,E2 -20641.374} C_VEL
LIN {X 0,Y 233.95,Z 293.636,A -85,B 0,C 180,E1 -20641.88,E2 -20641.88} C_VEL
LIN {X 0,Y 235.674,Z 254.63,A -85,B 0,C 180,E1 -20643.066,E2 -20643.066} C_VEL
LIN {X 0,Y 236.004,Z 244.138,A -85,B 0,C 180,E1 -20643.388,E2 -20643.388} C_VEL
LIN {X 0,Y 232.272,Z 222.357,A -85,B 0,C 180,E1 -20644.79,E2 -20644.79} C_VEL
LIN {X 0,Y 225.954,Z 207.518,A -85,B 0,C 180,E1 -20646.473,E2 -20646.473} C_VEL
LIN {X 0,Y 218.947,Z 193.485,A -85,B 0,C 180,E1 -20648.403,E2 -20648.403} C_VEL
LIN {X 0,Y 216.949,Z 189.894,A -85,B 0,C 180,E1 -20648.969,E2 -20648.969} C_VEL
LIN {X 0,Y 215.498,Z 186.68,A -85,B 0,C 180,E1 -20649.507,E2 -20649.507} C_VEL
LIN {X 0,Y 213.928,Z 180.387,A -85,B 0,C 180,E1 -20653.717,E2 -20653.717} C_VEL
LIN {X 0,Y 213.746,Z 179.355,A -85,B 0,C 180,E1 -20654.68,E2 -20654.68} C_VEL
LIN {X 0,Y 213.717,Z 179.347,A -85,B 0,C 180,E1 -20659.142,E2 -20659.142} C_VEL
LIN {X 0,Y 213.745,Z 179.349,A -85,B 0,C 180,E1 -20663.711,E2 -20663.711} C_VEL
LIN {X 0,Y 213.796,Z 179.352,A -85,B 0,C 180,E1 -20668.724,E2 -20668.724} C_VEL
LIN {X 0,Y 213.827,Z 179.314,A -85,B 0,C 180,E1 -20672.602,E2 -20672.602} C_VEL
LIN {X 0,Y 213.852,Z 179.346,A -85,B 0,C 180,E1 -20676.952,E2 -20676.952} C_VEL
LIN {X 0,Y 213.943,Z 179.299,A -85,B 0,C 180,E1 -20682.803,E2 -20682.803} C_VEL
LIN {X 0,Y 213.953,Z 179.326,A -85,B 0,C 180,E1 -20686.706,E2 -20686.706} C_VEL
LIN {X 0,Y 214.141,Z 179.261,A -85,B 0,C 180,E1 -20690.554,E2 -20690.554} C_VEL
LIN {X 0,Y 214.1,Z 179.312,A -85,B 0,C 180,E1 -20694.347,E2 -20694.347} C_VEL
LIN {X 0,Y 214.444,Z 179.24,A -85,B 0,C 180,E1 -20698.121,E2 -20698.121} C_VEL
LIN {X 0,Y 214.544,Z 179.21,A -85,B 0,C 180,E1 -20699.999,E2 -20699.999} C_VEL
LIN {X 0,Y 214.444,Z 179.235,A -85,B 0,C 180,E1 -20701.877,E2 -20701.877} C_VEL
LIN {X 0,Y 214.226,Z 179.274,A -85,B 0,C 180,E1 -20707.539,E2 -20707.539} C_VEL
LIN {X 0,Y 214.043,Z 179.284,A -85,B 0,C 180,E1 -20711.361,E2 -20711.361} C_VEL
LIN {X 0,Y 213.932,Z 179.336,A -85,B 0,C 180,E1 -20715.236,E2 -20715.236} C_VEL
LIN {X 0,Y 213.837,Z 179.305,A -85,B 0,C 180,E1 -20719.186,E2 -20719.186} C_VEL
LIN {X 0,Y 213.845,Z 179.348,A -85,B 0,C 180,E1 -20723.226,E2 -20723.226} C_VEL
LIN {X 0,Y 213.826,Z 179.315,A -85,B 0,C 180,E1 -20727.449,E2 -20727.449} C_VEL
LIN {X 0,Y 213.776,Z 179.355,A -85,B 0,C 180,E1 -20731.735,E2 -20731.735} C_VEL
LIN {X 0,Y 213.749,Z 179.344,A -85,B 0,C 180,E1 -20736.286,E2 -20736.286} C_VEL
LIN {X 0,Y 213.713,Z 179.343,A -85,B 0,C 180,E1 -20741.124,E2 -20741.124} C_VEL
LIN {X 0,Y 213.707,Z 179.364,A -85,B 0,C 180,E1 -20743.677,E2 -20743.677} C_VEL
LIN {X 0,Y 213.704,Z 179.306,A -85,B 0,C 180,E1 -20746.343,E2 -20746.343} C_VEL
LIN {X 0,Y 213.794,Z 179.504,A -85,B 0,C 180,E1 -20749.96,E2 -20749.96} C_VEL
LIN {X 0,Y 214.065,Z 180.639,A -85,B 0,C 180,E1 -20750.371,E2 -20750.371} C_VEL
LIN {X 0,Y 215.535,Z 183.211,A -85,B 0,C 180,E1 -20750.827,E2 -20750.827} C_VEL
LIN {X 0,Y 216.638,Z 184.741,A -85,B 0,C 180,E1 -20751.13,E2 -20751.13} C_VEL
LIN {X 0,Y 223.571,Z 195.904,A -85,B 0,C 180,E1 -20752.999,E2 -20752.999} C_VEL
LIN {X 0,Y 232.29,Z 211.801,A -85,B 0,C 180,E1 -20755.204,E2 -20755.204} C_VEL
LIN {X 0,Y 241.22,Z 229.429,A -85,B 0,C 180,E1 -20757.29,E2 -20757.29} C_VEL
LIN {X 0,Y 249.131,Z 241.76,A -85,B 0,C 180,E1 -20758.868,E2 -20758.868} C_VEL
LIN {X 0,Y 256.823,Z 251.792,A -85,B 0,C 180,E1 -20760.224,E2 -20760.224} C_VEL
LIN {X 0,Y 268.703,Z 265.025,A -85,B 0,C 180,E1 -20762.068,E2 -20762.068} C_VEL
LIN {X 0,Y 280.926,Z 276.676,A -85,B 0,C 180,E1 -20763.727,E2 -20763.727} C_VEL
LIN {X 0,Y 291.519,Z 285.752,A -85,B 0,C 180,E1 -20765.101,E2 -20765.101} C_VEL
LIN {X 0,Y 301.378,Z 293.765,A -85,B 0,C 180,E1 -20766.443,E2 -20766.443} C_VEL
LIN {X 0,Y 308.375,Z 299.126,A -85,B 0,C 180,E1 -20767.533,E2 -20767.533} C_VEL
LIN {X 0,Y 316.3,Z 305.023,A -85,B 0,C 180,E1 -20768.939,E2 -20768.939} C_VEL
LIN {X 0,Y 323.616,Z 310.447,A -85,B 0,C 180,E1 -20770.408,E2 -20770.408} C_VEL
LIN {X 0,Y 330.79,Z 315.404,A -85,B 0,C 180,E1 -20772.01,E2 -20772.01} C_VEL
LIN {X 0,Y 337.004,Z 319.931,A -85,B 0,C 180,E1 -20773.594,E2 -20773.594} C_VEL
LIN {X 0,Y 341.971,Z 323.311,A -85,B 0,C 180,E1 -20774.995,E2 -20774.995} C_VEL
LIN {X 0,Y 346.92,Z 326.251,A -85,B 0,C 180,E1 -20776.503,E2 -20776.503} C_VEL
LIN {X 0,Y 350.596,Z 328.598,A -85,B 0,C 180,E1 -20777.782,E2 -20777.782} C_VEL
LIN {X 0,Y 355.235,Z 332.022,A -85,B 0,C 180,E1 -20779.744,E2 -20779.744} C_VEL
LIN {X 0,Y 357.783,Z 333.589,A -85,B 0,C 180,E1 -20780.959,E2 -20780.959} C_VEL
LIN {X 0,Y 361.224,Z 335.46,A -85,B 0,C 180,E1 -20782.861,E2 -20782.861} C_VEL
LIN {X 0,Y 363.571,Z 336.524,A -85,B 0,C 180,E1 -20784.454,E2 -20784.454} C_VEL
LIN {X 0,Y 364.909,Z 337.057,A -85,B 0,C 180,E1 -20785.582,E2 -20785.582} C_VEL
LIN {X 0,Y 366.036,Z 337.399,A -85,B 0,C 180,E1 -20786.761,E2 -20786.761} C_VEL
LIN {X 0,Y 366.653,Z 337.726,A -85,B 0,C 180,E1 -20787.803,E2 -20787.803} C_VEL
LIN {X 0,Y 367.019,Z 337.987,A -85,B 0,C 180,E1 -20788.903,E2 -20788.903} C_VEL
LIN {X 0,Y 367.231,Z 337.908,A -85,B 0,C 180,E1 -20790,E2 -20790} C_VEL
LIN {X 0,Y 367.026,Z 337.961,A -85,B 0,C 180,E1 -20791.097,E2 -20791.097} C_VEL
LIN {X 0,Y 366.659,Z 337.695,A -85,B 0,C 180,E1 -20792.197,E2 -20792.197} C_VEL
LIN {X 0,Y 365.979,Z 337.352,A -85,B 0,C 180,E1 -20793.303,E2 -20793.303} C_VEL
LIN {X 0,Y 364.913,Z 337.021,A -85,B 0,C 180,E1 -20794.418,E2 -20794.418} C_VEL
LIN {X 0,Y 363.55,Z 336.525,A -85,B 0,C 180,E1 -20795.547,E2 -20795.547} C_VEL
LIN {X 0,Y 361.231,Z 335.471,A -85,B 0,C 180,E1 -20797.148,E2 -20797.148} C_VEL
LIN {X 0,Y 357.794,Z 333.544,A -85,B 0,C 180,E1 -20799.041,E2 -20799.041} C_VEL
LIN {X 0,Y 353.992,Z 331.113,A -85,B 0,C 180,E1 -20800.815,E2 -20800.815} C_VEL
LIN {X 0,Y 349.047,Z 327.486,A -85,B 0,C 180,E1 -20802.796,E2 -20802.796} C_VEL
LIN {X 0,Y 344.8,Z 325.05,A -85,B 0,C 180,E1 -20804.158,E2 -20804.158} C_VEL
LIN {X 0,Y 339.928,Z 321.981,A -85,B 0,C 180,E1 -20805.591,E2 -20805.591} C_VEL
LIN {X 0,Y 334.318,Z 317.92,A -85,B 0,C 180,E1 -20807.116,E2 -20807.116} C_VEL
LIN {X 0,Y 327.242,Z 313.068,A -85,B 0,C 180,E1 -20808.793,E2 -20808.793} C_VEL
LIN {X 0,Y 319.713,Z 307.507,A -85,B 0,C 180,E1 -20810.403,E2 -20810.403} C_VEL
LIN {X 0,Y 310.858,Z 301.068,A -85,B 0,C 180,E1 -20812.039,E2 -20812.039} C_VEL
LIN {X 0,Y 301.975,Z 294.216,A -85,B 0,C 180,E1 -20813.473,E2 -20813.473} C_VEL
LIN {X 0,Y 293.372,Z 287.286,A -85,B 0,C 180,E1 -20814.658,E2 -20814.658} C_VEL
LIN {X 0,Y 282.604,Z 278.17,A -85,B 0,C 180,E1 -20816.056,E2 -20816.056} C_VEL
LIN {X 0,Y 271.816,Z 268.058,A -85,B 0,C 180,E1 -20817.494,E2 -20817.494} C_VEL
LIN {X 0,Y 259.85,Z 255.375,A -85,B 0,C 180,E1 -20819.281,E2 -20819.281} C_VEL
LIN {X 0,Y 251.089,Z 244.528,A -85,B 0,C 180,E1 -20820.77,E2 -20820.77} C_VEL
LIN {X 0,Y 242.839,Z 232.139,A -85,B 0,C 180,E1 -20822.37,E2 -20822.37} C_VEL
LIN {X 0,Y 235.807,Z 219.08,A -85,B 0,C 180,E1 -20823.937,E2 -20823.937} C_VEL
LIN {X 0,Y 229.535,Z 206.57,A -85,B 0,C 180,E1 -20825.476,E2 -20825.476} C_VEL
LIN {X 0,Y 220.906,Z 191.428,A -85,B 0,C 180,E1 -20827.707,E2 -20827.707} C_VEL
LIN {X 0,Y 216.378,Z 184.182,A -85,B 0,C 180,E1 -20828.95,E2 -20828.95} C_VEL
LIN {X 0,Y 214.249,Z 181.149,A -85,B 0,C 180,E1 -20829.553,E2 -20829.553} C_VEL
LIN {X 0,Y 213.829,Z 179.771,A -85,B 0,C 180,E1 -20829.871,E2 -20829.871} C_VEL
LIN {X 0,Y 213.744,Z 179.361,A -85,B 0,C 180,E1 -20830.402,E2 -20830.402} C_VEL
LIN {X 0,Y 213.704,Z 179.307,A -85,B 0,C 180,E1 -20833.678,E2 -20833.678} C_VEL
LIN {X 0,Y 213.707,Z 179.365,A -85,B 0,C 180,E1 -20836.343,E2 -20836.343} C_VEL
LIN {X 0,Y 213.733,Z 179.355,A -85,B 0,C 180,E1 -20841.337,E2 -20841.337} C_VEL
LIN {X 0,Y 213.765,Z 179.33,A -85,B 0,C 180,E1 -20846.021,E2 -20846.021} C_VEL
LIN {X 0,Y 213.778,Z 179.341,A -85,B 0,C 180,E1 -20850.455,E2 -20850.455} C_VEL
LIN {X 0,Y 213.798,Z 179.334,A -85,B 0,C 180,E1 -20854.703,E2 -20854.703} C_VEL
LIN {X 0,Y 213.81,Z 179.327,A -85,B 0,C 180,E1 -20858.804,E2 -20858.804} C_VEL
LIN {X 0,Y 213.941,Z 179.306,A -85,B 0,C 180,E1 -20862.805,E2 -20862.805} C_VEL
LIN {X 0,Y 213.978,Z 179.323,A -85,B 0,C 180,E1 -20866.709,E2 -20866.709} C_VEL
LIN {X 0,Y 214.165,Z 179.26,A -85,B 0,C 180,E1 -20870.557,E2 -20870.557} C_VEL
LIN {X 0,Y 214.226,Z 179.274,A -85,B 0,C 180,E1 -20872.461,E2 -20872.461} C_VEL
LIN {X 0,Y 214.444,Z 179.235,A -85,B 0,C 180,E1 -20878.123,E2 -20878.123} C_VEL
LIN {X 0,Y 214.544,Z 179.21,A -85,B 0,C 180,E1 -20880.001,E2 -20880.001} C_VEL
LIN {X 0,Y 214.444,Z 179.24,A -85,B 0,C 180,E1 -20881.879,E2 -20881.879} C_VEL
LIN {X 0,Y 214.198,Z 179.272,A -85,B 0,C 180,E1 -20887.542,E2 -20887.542} C_VEL
LIN {X 0,Y 213.999,Z 179.291,A -85,B 0,C 180,E1 -20891.365,E2 -20891.365} C_VEL
LIN {X 0,Y 213.934,Z 179.328,A -85,B 0,C 180,E1 -20895.238,E2 -20895.238} C_VEL
LIN {X 0,Y 213.839,Z 179.303,A -85,B 0,C 180,E1 -20899.188,E2 -20899.188} C_VEL
LIN {X 0,Y 213.848,Z 179.345,A -85,B 0,C 180,E1 -20903.228,E2 -20903.228} C_VEL
LIN {X 0,Y 213.83,Z 179.314,A -85,B 0,C 180,E1 -20907.451,E2 -20907.451} C_VEL
LIN {X 0,Y 213.778,Z 179.349,A -85,B 0,C 180,E1 -20911.737,E2 -20911.737} C_VEL
LIN {X 0,Y 213.745,Z 179.349,A -85,B 0,C 180,E1 -20916.289,E2 -20916.289} C_VEL
LIN {X 0,Y 213.712,Z 179.349,A -85,B 0,C 180,E1 -20921.127,E2 -20921.127} C_VEL
LIN {X 0,Y 213.764,Z 179.527,A -85,B 0,C 180,E1 -20925.651,E2 -20925.651} C_VEL
LIN {X 0,Y 215.441,Z 186.51,A -85,B 0,C 180,E1 -20930.42,E2 -20930.42} C_VEL
LIN {X 0,Y 216.355,Z 188.766,A -85,B 0,C 180,E1 -20930.857,E2 -20930.857} C_VEL
LIN {X 0,Y 218.957,Z 193.52,A -85,B 0,C 180,E1 -20931.6,E2 -20931.6} C_VEL
LIN {X 0,Y 224.228,Z 203.864,A -85,B 0,C 180,E1 -20933.059,E2 -20933.059} C_VEL
LIN {X 0,Y 230.884,Z 218.902,A -85,B 0,C 180,E1 -20934.844,E2 -20934.844} C_VEL
LIN {X 0,Y 232.552,Z 223.537,A -85,B 0,C 180,E1 -20935.301,E2 -20935.301} C_VEL
LIN {X 0,Y 235.753,Z 242.698,A -85,B 0,C 180,E1 -20936.521,E2 -20936.521} C_VEL
LIN {X 0,Y 236.086,Z 245.577,A -85,B 0,C 180,E1 -20936.677,E2 -20936.677} C_VEL
LIN {X 0,Y 234.085,Z 292.683,A -85,B 0,C 180,E1 -20938.091,E2 -20938.091} C_VEL
LIN {X 0,Y 233.134,Z 303.176,A -85,B 0,C 180,E1 -20938.587,E2 -20938.587} C_VEL
LIN {X 0,Y 232.666,Z 307.332,A -85,B 0,C 180,E1 -20938.822,E2 -20938.822} C_VEL
LIN {X 0,Y 231.293,Z 312.955,A -85,B 0,C 180,E1 -20939.134,E2 -20939.134} C_VEL
LIN {X 0,Y 227.309,Z 321.882,A -85,B 0,C 180,E1 -20939.582,E2 -20939.582} C_VEL
LIN {X 0,Y 223.15,Z 330.627,A -85,B 0,C 180,E1 -20940.201,E2 -20940.201} C_VEL
LIN {X 0,Y 221.496,Z 335.678,A -85,B 0,C 180,E1 -20940.781,E2 -20940.781} C_VEL
LIN {X 0,Y 218.77,Z 346.38,A -85,B 0,C 180,E1 -20942.497,E2 -20942.497} C_VEL
LIN {X 0,Y 216.652,Z 354.121,A -85,B 0,C 180,E1 -20944.029,E2 -20944.029} C_VEL
LIN {X 0,Y 213.916,Z 363.255,A -85,B 0,C 180,E1 -20946.268,E2 -20946.268} C_VEL
LIN {X 0,Y 211.878,Z 369.873,A -85,B 0,C 180,E1 -20948.245,E2 -20948.245} C_VEL
LIN {X 0,Y 210.019,Z 375.995,A -85,B 0,C 180,E1 -20950.45,E2 -20950.45} C_VEL
LIN {X 0,Y 208.634,Z 380.498,A -85,B 0,C 180,E1 -20952.352,E2 -20952.352} C_VEL
LIN {X 0,Y 206.802,Z 385.987,A -85,B 0,C 180,E1 -20955.234,E2 -20955.234} C_VEL
LIN {X 0,Y 205.573,Z 390.316,A -85,B 0,C 180,E1 -20958.163,E2 -20958.163} C_VEL
LIN {X 0,Y 205.023,Z 392.687,A -85,B 0,C 180,E1 -20960.131,E2 -20960.131} C_VEL
LIN {X 0,Y 204.627,Z 394.489,A -85,B 0,C 180,E1 -20962.104,E2 -20962.104} C_VEL
LIN {X 0,Y 204.339,Z 396.945,A -85,B 0,C 180,E1 -20966.056,E2 -20966.056} C_VEL
LIN {X 0,Y 204.332,Z 397.538,A -85,B 0,C 180,E1 -20968.029,E2 -20968.029} C_VEL
LIN {X 0,Y 204.438,Z 397.696,A -85,B 0,C 180,E1 -20970,E2 -20970} C_VEL
LIN {X 0,Y 204.331,Z 397.538,A -85,B 0,C 180,E1 -20971.971,E2 -20971.971} C_VEL
LIN {X 0,Y 204.299,Z 396.944,A -85,B 0,C 180,E1 -20973.945,E2 -20973.945} C_VEL
LIN {X 0,Y 204.608,Z 394.489,A -85,B 0,C 180,E1 -20977.897,E2 -20977.897} C_VEL
LIN {X 0,Y 205.278,Z 391.535,A -85,B 0,C 180,E1 -20980.854,E2 -20980.854} C_VEL
LIN {X 0,Y 206.297,Z 387.541,A -85,B 0,C 180,E1 -20983.796,E2 -20983.796} C_VEL
LIN {X 0,Y 207.945,Z 382.412,A -85,B 0,C 180,E1 -20986.695,E2 -20986.695} C_VEL
LIN {X 0,Y 209.614,Z 377.149,A -85,B 0,C 180,E1 -20989.081,E2 -20989.081} C_VEL
LIN {X 0,Y 211.722,Z 370.836,A -85,B 0,C 180,E1 -20991.416,E2 -20991.416} C_VEL
LIN {X 0,Y 213.442,Z 364.882,A -85,B 0,C 180,E1 -20993.273,E2 -20993.273} C_VEL
LIN {X 0,Y 215.505,Z 357.957,A -85,B 0,C 180,E1 -20995.084,E2 -20995.084} C_VEL
LIN {X 0,Y 217.861,Z 349.783,A -85,B 0,C 180,E1 -20996.848,E2 -20996.848} C_VEL
LIN {X 0,Y 220.042,Z 341.274,A -85,B 0,C 180,E1 -20998.365,E2 -20998.365} C_VEL
LIN {X 0,Y 222.146,Z 332.565,A -85,B 0,C 180,E1 -20999.625,E2 -20999.625} C_VEL
LIN {X 0,Y 224.073,Z 322.809,A -85,B 0,C 180,E1 -21000.773,E2 -21000.773} C_VEL
LIN {X 0,Y 225.747,Z 312.731,A -85,B 0,C 180,E1 -21001.692,E2 -21001.692} C_VEL
LIN {X 0,Y 227.146,Z 302.484,A -85,B 0,C 180,E1 -21002.378,E2 -21002.378} C_VEL
LIN {X 0,Y 227.984,Z 293.087,A -85,B 0,C 180,E1 -21002.835,E2 -21002.835} C_VEL
LIN {X 0,Y 230.144,Z 246.378,A -85,B 0,C 180,E1 -21004.265,E2 -21004.265} C_VEL
LIN {X 0,Y 227.813,Z 231.087,A -85,B 0,C 180,E1 -21005.237,E2 -21005.237} C_VEL
LIN {X 0,Y 226.4,Z 224.363,A -85,B 0,C 180,E1 -21005.745,E2 -21005.745} C_VEL
LIN {X 0,Y 220.423,Z 210.391,A -85,B 0,C 180,E1 -21007.421,E2 -21007.421} C_VEL
LIN {X 0,Y 213.101,Z 195.536,A -85,B 0,C 180,E1 -21009.564,E2 -21009.564} C_VEL
LIN {X 0,Y 209.854,Z 189.977,A -85,B 0,C 180,E1 -21010.539,E2 -21010.539} C_VEL
LIN {X 0,Y 208.176,Z 186.471,A -85,B 0,C 180,E1 -21011.18,E2 -21011.18} C_VEL
LIN {X 0,Y 207.296,Z 182.913,A -85,B 0,C 180,E1 -21013.579,E2 -21013.579} C_VEL
LIN {X 0,Y 206.664,Z 180.247,A -85,B 0,C 180,E1 -21015.728,E2 -21015.728} C_VEL
LIN {X 0,Y 206.661,Z 180.223,A -85,B 0,C 180,E1 -21019.748,E2 -21019.748} C_VEL
LIN {X 0,Y 206.7,Z 180.213,A -85,B 0,C 180,E1 -21024.688,E2 -21024.688} C_VEL
LIN {X 0,Y 206.725,Z 180.236,A -85,B 0,C 180,E1 -21029.338,E2 -21029.338} C_VEL
LIN {X 0,Y 206.732,Z 180.198,A -85,B 0,C 180,E1 -21033.771,E2 -21033.771} C_VEL
LIN {X 0,Y 206.758,Z 180.221,A -85,B 0,C 180,E1 -21038.042,E2 -21038.042} C_VEL
LIN {X 0,Y 206.873,Z 180.172,A -85,B 0,C 180,E1 -21042.195,E2 -21042.195} C_VEL
LIN {X 0,Y 206.895,Z 180.209,A -85,B 0,C 180,E1 -21046.243,E2 -21046.243} C_VEL
LIN {X 0,Y 207.099,Z 180.137,A -85,B 0,C 180,E1 -21050.23,E2 -21050.23} C_VEL
LIN {X 0,Y 207.061,Z 180.188,A -85,B 0,C 180,E1 -21054.155,E2 -21054.155} C_VEL
LIN {X 0,Y 207.38,Z 180.119,A -85,B 0,C 180,E1 -21058.057,E2 -21058.057} C_VEL
LIN {X 0,Y 207.51,Z 180.086,A -85,B 0,C 180,E1 -21059.999,E2 -21059.999} C_VEL
LIN {X 0,Y 207.381,Z 180.114,A -85,B 0,C 180,E1 -21061.941,E2 -21061.941} C_VEL
LIN {X 0,Y 207.166,Z 180.147,A -85,B 0,C 180,E1 -21067.798,E2 -21067.798} C_VEL
LIN {X 0,Y 206.98,Z 180.168,A -85,B 0,C 180,E1 -21071.754,E2 -21071.754} C_VEL
LIN {X 0,Y 206.866,Z 180.21,A -85,B 0,C 180,E1 -21075.77,E2 -21075.77} C_VEL
LIN {X 0,Y 206.781,Z 180.186,A -85,B 0,C 180,E1 -21079.868,E2 -21079.868} C_VEL
LIN {X 0,Y 206.761,Z 180.228,A -85,B 0,C 180,E1 -21084.071,E2 -21084.071} C_VEL
LIN {X 0,Y 206.741,Z 180.201,A -85,B 0,C 180,E1 -21088.418,E2 -21088.418} C_VEL
LIN {X 0,Y 206.706,Z 180.217,A -85,B 0,C 180,E1 -21092.955,E2 -21092.955} C_VEL
LIN {X 0,Y 206.719,Z 180.209,A -85,B 0,C 180,E1 -21095.32,E2 -21095.32} C_VEL
LIN {X 0,Y 206.663,Z 180.22,A -85,B 0,C 180,E1 -21100.249,E2 -21100.249} C_VEL
LIN {X 0,Y 206.633,Z 180.224,A -85,B 0,C 180,E1 -21104.419,E2 -21104.419} C_VEL
LIN {X 0,Y 206.687,Z 180.418,A -85,B 0,C 180,E1 -21108.335,E2 -21108.335} C_VEL
LIN {X 0,Y 206.92,Z 181.32,A -85,B 0,C 180,E1 -21108.718,E2 -21108.718} C_VEL
LIN {X 0,Y 208.487,Z 184.105,A -85,B 0,C 180,E1 -21109.259,E2 -21109.259} C_VEL
LIN {X 0,Y 209.693,Z 185.656,A -85,B 0,C 180,E1 -21109.613,E2 -21109.613} C_VEL
LIN {X 0,Y 218.533,Z 199.712,A -85,B 0,C 180,E1 -21112.146,E2 -21112.146} C_VEL
LIN {X 0,Y 227.124,Z 215.592,A -85,B 0,C 180,E1 -21114.431,E2 -21114.431} C_VEL
LIN {X 0,Y 236.102,Z 233.545,A -85,B 0,C 180,E1 -21116.63,E2 -21116.63} C_VEL
LIN {X 0,Y 244.343,Z 246.489,A -85,B 0,C 180,E1 -21118.342,E2 -21118.342} C_VEL
LIN {X 0,Y 251.627,Z 256.094,A -85,B 0,C 180,E1 -21119.679,E2 -21119.679} C_VEL
LIN {X 0,Y 263.068,Z 269.071,A -85,B 0,C 180,E1 -21121.533,E2 -21121.533} C_VEL
LIN {X 0,Y 276.259,Z 281.873,A -85,B 0,C 180,E1 -21123.426,E2 -21123.426} C_VEL
LIN {X 0,Y 287.185,Z 291.348,A -85,B 0,C 180,E1 -21124.987,E2 -21124.987} C_VEL
LIN {X 0,Y 298.596,Z 300.539,A -85,B 0,C 180,E1 -21126.624,E2 -21126.624} C_VEL
LIN {X 0,Y 307.017,Z 307.017,A -85,B 0,C 180,E1 -21127.984,E2 -21127.984} C_VEL
LIN {X 0,Y 315.179,Z 312.902,A -85,B 0,C 180,E1 -21129.475,E2 -21129.475} C_VEL
LIN {X 0,Y 321.846,Z 317.919,A -85,B 0,C 180,E1 -21130.88,E2 -21130.88} C_VEL
LIN {X 0,Y 329.43,Z 323.058,A -85,B 0,C 180,E1 -21132.622,E2 -21132.622} C_VEL
LIN {X 0,Y 335.75,Z 327.723,A -85,B 0,C 180,E1 -21134.338,E2 -21134.338} C_VEL
LIN {X 0,Y 340.744,Z 330.857,A -85,B 0,C 180,E1 -21135.786,E2 -21135.786} C_VEL
LIN {X 0,Y 345.687,Z 333.761,A -85,B 0,C 180,E1 -21137.383,E2 -21137.383} C_VEL
LIN {X 0,Y 350.428,Z 337.29,A -85,B 0,C 180,E1 -21139.329,E2 -21139.329} C_VEL
LIN {X 0,Y 355.179,Z 340.285,A -85,B 0,C 180,E1 -21141.63,E2 -21141.63} C_VEL
LIN {X 0,Y 357.985,Z 341.688,A -85,B 0,C 180,E1 -21143.235,E2 -21143.235} C_VEL
LIN {X 0,Y 359.991,Z 342.605,A -85,B 0,C 180,E1 -21144.651,E2 -21144.651} C_VEL
LIN {X 0,Y 362.118,Z 343.338,A -85,B 0,C 180,E1 -21146.662,E2 -21146.662} C_VEL
LIN {X 0,Y 362.819,Z 343.683,A -85,B 0,C 180,E1 -21147.78,E2 -21147.78} C_VEL
LIN {X 0,Y 363.186,Z 343.955,A -85,B 0,C 180,E1 -21148.891,E2 -21148.891} C_VEL
LIN {X 0,Y 363.418,Z 343.882,A -85,B 0,C 180,E1 -21150,E2 -21150} C_VEL
LIN {X 0,Y 363.197,Z 343.923,A -85,B 0,C 180,E1 -21151.109,E2 -21151.109} C_VEL
LIN {X 0,Y 362.824,Z 343.649,A -85,B 0,C 180,E1 -21152.22,E2 -21152.22} C_VEL
LIN {X 0,Y 362.117,Z 343.302,A -85,B 0,C 180,E1 -21153.338,E2 -21153.338} C_VEL
LIN {X 0,Y 359.987,Z 342.596,A -85,B 0,C 180,E1 -21155.342,E2 -21155.342} C_VEL
LIN {X 0,Y 357.952,Z 341.703,A -85,B 0,C 180,E1 -21156.765,E2 -21156.765} C_VEL
LIN {X 0,Y 355.193,Z 340.255,A -85,B 0,C 180,E1 -21158.386,E2 -21158.386} C_VEL
LIN {X 0,Y 350.424,Z 337.272,A -85,B 0,C 180,E1 -21160.668,E2 -21160.668} C_VEL
LIN {X 0,Y 345.669,Z 333.791,A -85,B 0,C 180,E1 -21162.604,E2 -21162.604} C_VEL
LIN {X 0,Y 340.279,Z 330.582,A -85,B 0,C 180,E1 -21164.35,E2 -21164.35} C_VEL
LIN {X 0,Y 335.204,Z 327.328,A -85,B 0,C 180,E1 -21165.817,E2 -21165.817} C_VEL
LIN {X 0,Y 329.355,Z 323.068,A -85,B 0,C 180,E1 -21167.382,E2 -21167.382} C_VEL
LIN {X 0,Y 321.812,Z 317.933,A -85,B 0,C 180,E1 -21169.122,E2 -21169.122} C_VEL
LIN {X 0,Y 315.169,Z 312.922,A -85,B 0,C 180,E1 -21170.52,E2 -21170.52} C_VEL
LIN {X 0,Y 307.009,Z 307.045,A -85,B 0,C 180,E1 -21172.012,E2 -21172.012} C_VEL
LIN {X 0,Y 298.591,Z 300.533,A -85,B 0,C 180,E1 -21173.374,E2 -21173.374} C_VEL
LIN {X 0,Y 287.551,Z 291.647,A -85,B 0,C 180,E1 -21174.962,E2 -21174.962} C_VEL
LIN {X 0,Y 278.081,Z 283.494,A -85,B 0,C 180,E1 -21176.312,E2 -21176.312} C_VEL
LIN {X 0,Y 268.004,Z 274.004,A -85,B 0,C 180,E1 -21177.745,E2 -21177.745} C_VEL
LIN {X 0,Y 255.271,Z 260.489,A -85,B 0,C 180,E1 -21179.7,E2 -21179.7} C_VEL
LIN {X 0,Y 246.218,Z 249.158,A -85,B 0,C 180,E1 -21181.298,E2 -21181.298} C_VEL
LIN {X 0,Y 237.886,Z 236.535,A -85,B 0,C 180,E1 -21182.98,E2 -21182.98} C_VEL
LIN {X 0,Y 230.527,Z 222.681,A -85,B 0,C 180,E1 -21184.698,E2 -21184.698} C_VEL
LIN {X 0,Y 224.663,Z 210.87,A -85,B 0,C 180,E1 -21186.205,E2 -21186.205} C_VEL
LIN {X 0,Y 216.432,Z 196.199,A -85,B 0,C 180,E1 -21188.437,E2 -21188.437} C_VEL
LIN {X 0,Y 210.761,Z 187.483,A -85,B 0,C 180,E1 -21190.059,E2 -21190.059} C_VEL
LIN {X 0,Y 209.03,Z 184.657,A -85,B 0,C 180,E1 -21190.588,E2 -21190.588} C_VEL
LIN {X 0,Y 207.196,Z 182.096,A -85,B 0,C 180,E1 -21191.15,E2 -21191.15} C_VEL
LIN {X 0,Y 206.757,Z 180.766,A -85,B 0,C 180,E1 -21191.453,E2 -21191.453} C_VEL
LIN {X 0,Y 206.619,Z 180.221,A -85,B 0,C 180,E1 -21192.134,E2 -21192.134} C_VEL
LIN {X 0,Y 206.633,Z 180.224,A -85,B 0,C 180,E1 -21195.581,E2 -21195.581} C_VEL
LIN {X 0,Y 206.663,Z 180.22,A -85,B 0,C 180,E1 -21199.751,E2 -21199.751} C_VEL
LIN {X 0,Y 206.728,Z 180.208,A -85,B 0,C 180,E1 -21204.696,E2 -21204.696} C_VEL
LIN {X 0,Y 206.721,Z 180.236,A -85,B 0,C 180,E1 -21209.34,E2 -21209.34} C_VEL
LIN {X 0,Y 206.729,Z 180.202,A -85,B 0,C 180,E1 -21213.773,E2 -21213.773} C_VEL
LIN {X 0,Y 206.755,Z 180.219,A -85,B 0,C 180,E1 -21218.044,E2 -21218.044} C_VEL
LIN {X 0,Y 206.871,Z 180.178,A -85,B 0,C 180,E1 -21222.198,E2 -21222.198} C_VEL
LIN {X 0,Y 206.912,Z 180.208,A -85,B 0,C 180,E1 -21226.247,E2 -21226.247} C_VEL
LIN {X 0,Y 207.104,Z 180.138,A -85,B 0,C 180,E1 -21230.232,E2 -21230.232} C_VEL
LIN {X 0,Y 207.166,Z 180.147,A -85,B 0,C 180,E1 -21232.202,E2 -21232.202} C_VEL
LIN {X 0,Y 207.381,Z 180.114,A -85,B 0,C 180,E1 -21238.059,E2 -21238.059} C_VEL
LIN {X 0,Y 207.51,Z 180.086,A -85,B 0,C 180,E1 -21240.001,E2 -21240.001} C_VEL
LIN {X 0,Y 207.38,Z 180.119,A -85,B 0,C 180,E1 -21241.943,E2 -21241.943} C_VEL
LIN {X 0,Y 207.14,Z 180.145,A -85,B 0,C 180,E1 -21247.801,E2 -21247.801} C_VEL
LIN {X 0,Y 206.924,Z 180.176,A -85,B 0,C 180,E1 -21251.759,E2 -21251.759} C_VEL
LIN {X 0,Y 206.867,Z 180.201,A -85,B 0,C 180,E1 -21255.772,E2 -21255.772} C_VEL
LIN {X 0,Y 206.783,Z 180.186,A -85,B 0,C 180,E1 -21259.87,E2 -21259.87} C_VEL
LIN {X 0,Y 206.764,Z 180.22,A -85,B 0,C 180,E1 -21264.073,E2 -21264.073} C_VEL
LIN {X 0,Y 206.745,Z 180.203,A -85,B 0,C 180,E1 -21268.42,E2 -21268.42} C_VEL
LIN {X 0,Y 206.703,Z 180.213,A -85,B 0,C 180,E1 -21272.958,E2 -21272.958} C_VEL
LIN {X 0,Y 206.683,Z 180.239,A -85,B 0,C 180,E1 -21277.74,E2 -21277.74} C_VEL
LIN {X 0,Y 206.642,Z 180.233,A -85,B 0,C 180,E1 -21281.563,E2 -21281.563} C_VEL
LIN {X 0,Y 206.682,Z 180.341,A -85,B 0,C 180,E1 -21284.433,E2 -21284.433} C_VEL
LIN {X 0,Y 208.091,Z 186.263,A -85,B 0,C 180,E1 -21288.725,E2 -21288.725} C_VEL
LIN {X 0,Y 208.973,Z 188.448,A -85,B 0,C 180,E1 -21289.187,E2 -21289.187} C_VEL
LIN {X 0,Y 211.634,Z 193.003,A -85,B 0,C 180,E1 -21290,E2 -21290} C_VEL
LIN {X 0,Y 217.583,Z 204.3,A -85,B 0,C 180,E1 -21291.759,E2 -21291.759} C_VEL
LIN {X 0,Y 225.075,Z 221.046,A -85,B 0,C 180,E1 -21293.886,E2 -21293.886} C_VEL
LIN {X 0,Y 226.948,Z 226.063,A -85,B 0,C 180,E1 -21294.419,E2 -21294.419} C_VEL
LIN {X 0,Y 230.106,Z 245.763,A -85,B 0,C 180,E1 -21295.706,E2 -21295.706} C_VEL
LIN {X 0,Y 228.051,Z 293.189,A -85,B 0,C 180,E1 -21297.178,E2 -21297.178} C_VEL
LIN {X 0,Y 226.925,Z 304.646,A -85,B 0,C 180,E1 -21297.749,E2 -21297.749} C_VEL
LIN {X 0,Y 224.99,Z 317.755,A -85,B 0,C 180,E1 -21298.714,E2 -21298.714} C_VEL
LIN {X 0,Y 222.803,Z 329.301,A -85,B 0,C 180,E1 -21299.95,E2 -21299.95} C_VEL
LIN {X 0,Y 221.496,Z 335.678,A -85,B 0,C 180,E1 -21300.781,E2 -21300.781} C_VEL
LIN {X 0,Y 219.761,Z 340.758,A -85,B 0,C 180,E1 -21301.426,E2 -21301.426} C_VEL
LIN {X 0,Y 215.101,Z 348.624,A -85,B 0,C 180,E1 -21302.449,E2 -21302.449} C_VEL
LIN {X 0,Y 210.288,Z 355.962,A -85,B 0,C 180,E1 -21303.698,E2 -21303.698} C_VEL
LIN {X 0,Y 208.348,Z 360.212,A -85,B 0,C 180,E1 -21304.689,E2 -21304.689} C_VEL
LIN {X 0,Y 205.364,Z 369.402,A -85,B 0,C 180,E1 -21307.41,E2 -21307.41} C_VEL
LIN {X 0,Y 203.338,Z 375.803,A -85,B 0,C 180,E1 -21309.78,E2 -21309.78} C_VEL
LIN {X 0,Y 201.841,Z 380.305,A -85,B 0,C 180,E1 -21311.737,E2 -21311.737} C_VEL
LIN {X 0,Y 199.903,Z 385.795,A -85,B 0,C 180,E1 -21314.712,E2 -21314.712} C_VEL
LIN {X 0,Y 198.597,Z 390.123,A -85,B 0,C 180,E1 -21317.741,E2 -21317.741} C_VEL
LIN {X 0,Y 198,Z 392.494,A -85,B 0,C 180,E1 -21319.777,E2 -21319.777} C_VEL
LIN {X 0,Y 197.578,Z 394.297,A -85,B 0,C 180,E1 -21321.82,E2 -21321.82} C_VEL
LIN {X 0,Y 197.247,Z 396.803,A -85,B 0,C 180,E1 -21326.086,E2 -21326.086} C_VEL
LIN {X 0,Y 197.241,Z 397.346,A -85,B 0,C 180,E1 -21327.958,E2 -21327.958} C_VEL
LIN {X 0,Y 197.34,Z 397.504,A -85,B 0,C 180,E1 -21330,E2 -21330} C_VEL
LIN {X 0,Y 197.237,Z 397.346,A -85,B 0,C 180,E1 -21332.042,E2 -21332.042} C_VEL
LIN {X 0,Y 197.21,Z 396.752,A -85,B 0,C 180,E1 -21334.087,E2 -21334.087} C_VEL
LIN {X 0,Y 197.544,Z 394.296,A -85,B 0,C 180,E1 -21338.181,E2 -21338.181} C_VEL
LIN {X 0,Y 198.268,Z 391.342,A -85,B 0,C 180,E1 -21341.242,E2 -21341.242} C_VEL
LIN {X 0,Y 199.373,Z 387.349,A -85,B 0,C 180,E1 -21344.285,E2 -21344.285} C_VEL
LIN {X 0,Y 201.132,Z 382.22,A -85,B 0,C 180,E1 -21347.278,E2 -21347.278} C_VEL
LIN {X 0,Y 202.899,Z 376.957,A -85,B 0,C 180,E1 -21349.738,E2 -21349.738} C_VEL
LIN {X 0,Y 205.067,Z 370.643,A -85,B 0,C 180,E1 -21352.147,E2 -21352.147} C_VEL
LIN {X 0,Y 207.411,Z 363.063,A -85,B 0,C 180,E1 -21354.524,E2 -21354.524} C_VEL
LIN {X 0,Y 210.297,Z 353.93,A -85,B 0,C 180,E1 -21356.818,E2 -21356.818} C_VEL
LIN {X 0,Y 213.47,Z 342.433,A -85,B 0,C 180,E1 -21359.052,E2 -21359.052} C_VEL
LIN {X 0,Y 215.986,Z 332.373,A -85,B 0,C 180,E1 -21360.558,E2 -21360.558} C_VEL
LIN {X 0,Y 217.806,Z 323.624,A -85,B 0,C 180,E1 -21361.624,E2 -21361.624} C_VEL
LIN {X 0,Y 219.55,Z 313.827,A -85,B 0,C 180,E1 -21362.56,E2 -21362.56} C_VEL
LIN {X 0,Y 221.077,Z 303.265,A -85,B 0,C 180,E1 -21363.305,E2 -21363.305} C_VEL
LIN {X 0,Y 222.057,Z 292.654,A -85,B 0,C 180,E1 -21363.84,E2 -21363.84} C_VEL
LIN {X 0,Y 224.194,Z 246.352,A -85,B 0,C 180,E1 -21365.301,E2 -21365.301} C_VEL
LIN {X 0,Y 221.222,Z 227.987,A -85,B 0,C 180,E1 -21366.566,E2 -21366.566} C_VEL
LIN {X 0,Y 215.28,Z 213.907,A -85,B 0,C 180,E1 -21368.322,E2 -21368.322} C_VEL
LIN {X 0,Y 208.396,Z 199.83,A -85,B 0,C 180,E1 -21370.443,E2 -21370.443} C_VEL
LIN {X 0,Y 202.961,Z 190.308,A -85,B 0,C 180,E1 -21372.198,E2 -21372.198} C_VEL
LIN {X 0,Y 200.859,Z 186.279,A -85,B 0,C 180,E1 -21373.019,E2 -21373.019} C_VEL
LIN {X 0,Y 200.345,Z 183.959,A -85,B 0,C 180,E1 -21374.554,E2 -21374.554} C_VEL
LIN {X 0,Y 199.625,Z 181.165,A -85,B 0,C 180,E1 -21376.895,E2 -21376.895} C_VEL
LIN {X 0,Y 199.612,Z 181.103,A -85,B 0,C 180,E1 -21380.767,E2 -21380.767} C_VEL
LIN {X 0,Y 199.614,Z 181.09,A -85,B 0,C 180,E1 -21385.713,E2 -21385.713} C_VEL
LIN {X 0,Y 199.702,Z 181.099,A -85,B 0,C 180,E1 -21388.136,E2 -21388.136} C_VEL
LIN {X 0,Y 199.687,Z 181.073,A -85,B 0,C 180,E1 -21392.771,E2 -21392.771} C_VEL
LIN {X 0,Y 199.739,Z 181.102,A -85,B 0,C 180,E1 -21397.228,E2 -21397.228} C_VEL
LIN {X 0,Y 199.796,Z 181.051,A -85,B 0,C 180,E1 -21401.757,E2 -21401.757} C_VEL
LIN {X 0,Y 199.836,Z 181.089,A -85,B 0,C 180,E1 -21405.747,E2 -21405.747} C_VEL
LIN {X 0,Y 200.022,Z 181.018,A -85,B 0,C 180,E1 -21409.881,E2 -21409.881} C_VEL
LIN {X 0,Y 200.022,Z 181.061,A -85,B 0,C 180,E1 -21413.948,E2 -21413.948} C_VEL
LIN {X 0,Y 200.32,Z 180.998,A -85,B 0,C 180,E1 -21417.988,E2 -21417.988} C_VEL
LIN {X 0,Y 200.475,Z 180.961,A -85,B 0,C 180,E1 -21419.999,E2 -21419.999} C_VEL
LIN {X 0,Y 200.031,Z 181.063,A -85,B 0,C 180,E1 -21424.028,E2 -21424.028} C_VEL
LIN {X 0,Y 200.11,Z 181.021,A -85,B 0,C 180,E1 -21428.075,E2 -21428.075} C_VEL
LIN {X 0,Y 199.912,Z 181.053,A -85,B 0,C 180,E1 -21432.176,E2 -21432.176} C_VEL
LIN {X 0,Y 199.803,Z 181.079,A -85,B 0,C 180,E1 -21436.342,E2 -21436.342} C_VEL
LIN {X 0,Y 199.697,Z 181.074,A -85,B 0,C 180,E1 -21440.604,E2 -21440.604} C_VEL
LIN {X 0,Y 199.67,Z 181.097,A -85,B 0,C 180,E1 -21444.983,E2 -21444.983} C_VEL
LIN {X 0,Y 199.672,Z 181.095,A -85,B 0,C 180,E1 -21449.521,E2 -21449.521} C_VEL
LIN {X 0,Y 199.661,Z 181.102,A -85,B 0,C 180,E1 -21452.351,E2 -21452.351} C_VEL
LIN {X 0,Y 199.637,Z 181.108,A -85,B 0,C 180,E1 -21456.759,E2 -21456.759} C_VEL
LIN {X 0,Y 199.636,Z 181.101,A -85,B 0,C 180,E1 -21459.32,E2 -21459.32} C_VEL
LIN {X 0,Y 199.578,Z 181.091,A -85,B 0,C 180,E1 -21464.77,E2 -21464.77} C_VEL
LIN {X 0,Y 199.624,Z 181.441,A -85,B 0,C 180,E1 -21466.634,E2 -21466.634} C_VEL
LIN {X 0,Y 200.027,Z 182.793,A -85,B 0,C 180,E1 -21467.047,E2 -21467.047} C_VEL
LIN {X 0,Y 201.773,Z 185.399,A -85,B 0,C 180,E1 -21467.645,E2 -21467.645} C_VEL
LIN {X 0,Y 202.806,Z 186.739,A -85,B 0,C 180,E1 -21467.976,E2 -21467.976} C_VEL
LIN {X 0,Y 208.212,Z 195.028,A -85,B 0,C 180,E1 -21469.681,E2 -21469.681} C_VEL
LIN {X 0,Y 214.352,Z 205.064,A -85,B 0,C 180,E1 -21471.492,E2 -21471.492} C_VEL
LIN {X 0,Y 222.282,Z 219.92,A -85,B 0,C 180,E1 -21473.698,E2 -21473.698} C_VEL
LIN {X 0,Y 231.174,Z 237.904,A -85,B 0,C 180,E1 -21475.976,E2 -21475.976} C_VEL
LIN {X 0,Y 239.547,Z 251.159,A -85,B 0,C 180,E1 -21477.79,E2 -21477.79} C_VEL
LIN {X 0,Y 247.018,Z 261.106,A -85,B 0,C 180,E1 -21479.214,E2 -21479.214} C_VEL
LIN {X 0,Y 258.712,Z 274.429,A -85,B 0,C 180,E1 -21481.171,E2 -21481.171} C_VEL
LIN {X 0,Y 271.137,Z 286.73,A -85,B 0,C 180,E1 -21483.102,E2 -21483.102} C_VEL
LIN {X 0,Y 282.578,Z 296.73,A -85,B 0,C 180,E1 -21484.885,E2 -21484.885} C_VEL
LIN {X 0,Y 295.698,Z 307.176,A -85,B 0,C 180,E1 -21486.895,E2 -21486.895} C_VEL
LIN {X 0,Y 304.238,Z 313.765,A -85,B 0,C 180,E1 -21488.309,E2 -21488.309} C_VEL
LIN {X 0,Y 312.287,Z 319.626,A -85,B 0,C 180,E1 -21489.815,E2 -21489.815} C_VEL
LIN {X 0,Y 319.101,Z 324.612,A -85,B 0,C 180,E1 -21491.269,E2 -21491.269} C_VEL
LIN {X 0,Y 325.892,Z 329.251,A -85,B 0,C 180,E1 -21492.86,E2 -21492.86} C_VEL
LIN {X 0,Y 331.707,Z 333.531,A -85,B 0,C 180,E1 -21494.449,E2 -21494.449} C_VEL
LIN {X 0,Y 337.778,Z 337.296,A -85,B 0,C 180,E1 -21496.231,E2 -21496.231} C_VEL
LIN {X 0,Y 341.104,Z 339.213,A -85,B 0,C 180,E1 -21497.308,E2 -21497.308} C_VEL
LIN {X 0,Y 344.195,Z 341.554,A -85,B 0,C 180,E1 -21498.545,E2 -21498.545} C_VEL
LIN {X 0,Y 346.39,Z 343.086,A -85,B 0,C 180,E1 -21499.479,E2 -21499.479} C_VEL
LIN {X 0,Y 349.07,Z 344.847,A -85,B 0,C 180,E1 -21500.731,E2 -21500.731} C_VEL
LIN {X 0,Y 351.412,Z 346.234,A -85,B 0,C 180,E1 -21501.953,E2 -21501.953} C_VEL
LIN {X 0,Y 353.797,Z 347.39,A -85,B 0,C 180,E1 -21503.319,E2 -21503.319} C_VEL
LIN {X 0,Y 355.263,Z 348.068,A -85,B 0,C 180,E1 -21504.324,E2 -21504.324} C_VEL
LIN {X 0,Y 356.689,Z 348.663,A -85,B 0,C 180,E1 -21505.48,E2 -21505.48} C_VEL
LIN {X 0,Y 357.83,Z 349.014,A -85,B 0,C 180,E1 -21506.622,E2 -21506.622} C_VEL
LIN {X 0,Y 358.656,Z 349.422,A -85,B 0,C 180,E1 -21507.934,E2 -21507.934} C_VEL
LIN {X 0,Y 359.163,Z 349.57,A -85,B 0,C 180,E1 -21510,E2 -21510} C_VEL
LIN {X 0,Y 358.653,Z 349.386,A -85,B 0,C 180,E1 -21512.05,E2 -21512.05} C_VEL
LIN {X 0,Y 357.819,Z 348.99,A -85,B 0,C 180,E1 -21513.378,E2 -21513.378} C_VEL
LIN {X 0,Y 356.672,Z 348.64,A -85,B 0,C 180,E1 -21514.521,E2 -21514.521} C_VEL
LIN {X 0,Y 355.235,Z 348.057,A -85,B 0,C 180,E1 -21515.677,E2 -21515.677} C_VEL
LIN {X 0,Y 353.464,Z 347.266,A -85,B 0,C 180,E1 -21516.852,E2 -21516.852} C_VEL
LIN {X 0,Y 351.413,Z 346.204,A -85,B 0,C 180,E1 -21518.047,E2 -21518.047} C_VEL
LIN {X 0,Y 348.976,Z 344.731,A -85,B 0,C 180,E1 -21519.322,E2 -21519.322} C_VEL
LIN {X 0,Y 346.378,Z 343.069,A -85,B 0,C 180,E1 -21520.522,E2 -21520.522} C_VEL
LIN {X 0,Y 343.319,Z 340.889,A -85,B 0,C 180,E1 -21521.812,E2 -21521.812} C_VEL
LIN {X 0,Y 339.373,Z 338.215,A -85,B 0,C 180,E1 -21523.27,E2 -21523.27} C_VEL
LIN {X 0,Y 334.361,Z 335.222,A -85,B 0,C 180,E1 -21524.79,E2 -21524.79} C_VEL
LIN {X 0,Y 327.962,Z 330.837,A -85,B 0,C 180,E1 -21526.587,E2 -21526.587} C_VEL
LIN {X 0,Y 321.721,Z 326.377,A -85,B 0,C 180,E1 -21528.148,E2 -21528.148} C_VEL
LIN {X 0,Y 313.828,Z 320.889,A -85,B 0,C 180,E1 -21529.856,E2 -21529.856} C_VEL
LIN {X 0,Y 308.491,Z 316.802,A -85,B 0,C 180,E1 -21530.926,E2 -21530.926} C_VEL
LIN {X 0,Y 300.204,Z 310.745,A -85,B 0,C 180,E1 -21532.375,E2 -21532.375} C_VEL
LIN {X 0,Y 290.245,Z 303.085,A -85,B 0,C 180,E1 -21533.927,E2 -21533.927} C_VEL
LIN {X 0,Y 275.776,Z 290.932,A -85,B 0,C 180,E1 -21536.167,E2 -21536.167} C_VEL
LIN {X 0,Y 265.216,Z 281.026,A -85,B 0,C 180,E1 -21537.823,E2 -21537.823} C_VEL
LIN {X 0,Y 251.905,Z 266.977,A -85,B 0,C 180,E1 -21539.932,E2 -21539.932} C_VEL
LIN {X 0,Y 241.983,Z 254.621,A -85,B 0,C 180,E1 -21541.727,E2 -21541.727} C_VEL
LIN {X 0,Y 234.012,Z 242.649,A -85,B 0,C 180,E1 -21543.381,E2 -21543.381} C_VEL
LIN {X 0,Y 226.841,Z 229.587,A -85,B 0,C 180,E1 -21545.087,E2 -21545.087} C_VEL
LIN {X 0,Y 219.869,Z 215.231,A -85,B 0,C 180,E1 -21546.956,E2 -21546.956} C_VEL
LIN {X 0,Y 212.137,Z 201.171,A -85,B 0,C 180,E1 -21549.156,E2 -21549.156} C_VEL
LIN {X 0,Y 204.456,Z 189.29,A -85,B 0,C 180,E1 -21551.489,E2 -21551.489} C_VEL
LIN {X 0,Y 201.947,Z 185.557,A -85,B 0,C 180,E1 -21552.302,E2 -21552.302} C_VEL
LIN {X 0,Y 200.138,Z 183.051,A -85,B 0,C 180,E1 -21552.904,E2 -21552.904} C_VEL
LIN {X 0,Y 199.679,Z 181.621,A -85,B 0,C 180,E1 -21553.259,E2 -21553.259} C_VEL
LIN {X 0,Y 199.594,Z 181.195,A -85,B 0,C 180,E1 -21553.645,E2 -21553.645} C_VEL
LIN {X 0,Y 199.58,Z 181.108,A -85,B 0,C 180,E1 -21558.007,E2 -21558.007} C_VEL
LIN {X 0,Y 199.638,Z 181.102,A -85,B 0,C 180,E1 -21560.757,E2 -21560.757} C_VEL
LIN {X 0,Y 199.631,Z 181.089,A -85,B 0,C 180,E1 -21565.719,E2 -21565.719} C_VEL
LIN {X 0,Y 199.701,Z 181.106,A -85,B 0,C 180,E1 -21568.138,E2 -21568.138} C_VEL
LIN {X 0,Y 199.683,Z 181.075,A -85,B 0,C 180,E1 -21572.773,E2 -21572.773} C_VEL
LIN {X 0,Y 199.736,Z 181.104,A -85,B 0,C 180,E1 -21577.23,E2 -21577.23} C_VEL
LIN {X 0,Y 199.794,Z 181.055,A -85,B 0,C 180,E1 -21581.759,E2 -21581.759} C_VEL
LIN {X 0,Y 199.846,Z 181.092,A -85,B 0,C 180,E1 -21585.75,E2 -21585.75} C_VEL
LIN {X 0,Y 200.069,Z 181.014,A -85,B 0,C 180,E1 -21589.885,E2 -21589.885} C_VEL
LIN {X 0,Y 200.034,Z 181.063,A -85,B 0,C 180,E1 -21593.951,E2 -21593.951} C_VEL
LIN {X 0,Y 200.321,Z 180.993,A -85,B 0,C 180,E1 -21597.991,E2 -21597.991} C_VEL
LIN {X 0,Y 200.475,Z 180.961,A -85,B 0,C 180,E1 -21600.001,E2 -21600.001} C_VEL
LIN {X 0,Y 200.027,Z 181.066,A -85,B 0,C 180,E1 -21604.031,E2 -21604.031} C_VEL
LIN {X 0,Y 200.088,Z 181.019,A -85,B 0,C 180,E1 -21608.078,E2 -21608.078} C_VEL
LIN {X 0,Y 199.874,Z 181.06,A -85,B 0,C 180,E1 -21612.18,E2 -21612.18} C_VEL
LIN {X 0,Y 199.805,Z 181.07,A -85,B 0,C 180,E1 -21616.345,E2 -21616.345} C_VEL
LIN {X 0,Y 199.7,Z 181.075,A -85,B 0,C 180,E1 -21620.606,E2 -21620.606} C_VEL
LIN {X 0,Y 199.673,Z 181.089,A -85,B 0,C 180,E1 -21624.985,E2 -21624.985} C_VEL
LIN {X 0,Y 199.676,Z 181.1,A -85,B 0,C 180,E1 -21629.523,E2 -21629.523} C_VEL
LIN {X 0,Y 199.679,Z 181.094,A -85,B 0,C 180,E1 -21632.359,E2 -21632.359} C_VEL
LIN {X 0,Y 199.625,Z 181.114,A -85,B 0,C 180,E1 -21636.764,E2 -21636.764} C_VEL
LIN {X 0,Y 199.609,Z 181.102,A -85,B 0,C 180,E1 -21639.329,E2 -21639.329} C_VEL
LIN {X 0,Y 199.646,Z 181.275,A -85,B 0,C 180,E1 -21643.263,E2 -21643.263} C_VEL
LIN {X 0,Y 200.809,Z 186.11,A -85,B 0,C 180,E1 -21646.918,E2 -21646.918} C_VEL
LIN {X 0,Y 202.645,Z 189.859,A -85,B 0,C 180,E1 -21647.701,E2 -21647.701} C_VEL
LIN {X 0,Y 204.203,Z 192.4,A -85,B 0,C 180,E1 -21648.212,E2 -21648.212} C_VEL
LIN {X 0,Y 209.174,Z 201.352,A -85,B 0,C 180,E1 -21649.804,E2 -21649.804} C_VEL
LIN {X 0,Y 215.132,Z 213.582,A -85,B 0,C 180,E1 -21651.633,E2 -21651.633} C_VEL
LIN {X 0,Y 221.367,Z 228.42,A -85,B 0,C 180,E1 -21653.479,E2 -21653.479} C_VEL
LIN {X 0,Y 224.256,Z 247.431,A -85,B 0,C 180,E1 -21654.752,E2 -21654.752} C_VEL
LIN {X 0,Y 222.157,Z 292.725,A -85,B 0,C 180,E1 -21656.177,E2 -21656.177} C_VEL
LIN {X 0,Y 221.03,Z 303.956,A -85,B 0,C 180,E1 -21656.741,E2 -21656.741} C_VEL
LIN {X 0,Y 219.168,Z 316.4,A -85,B 0,C 180,E1 -21657.649,E2 -21657.649} C_VEL
LIN {X 0,Y 216.666,Z 329.109,A -85,B 0,C 180,E1 -21659.007,E2 -21659.007} C_VEL
LIN {X 0,Y 214.58,Z 338.383,A -85,B 0,C 180,E1 -21660.306,E2 -21660.306} C_VEL
LIN {X 0,Y 212.167,Z 347.323,A -85,B 0,C 180,E1 -21661.834,E2 -21661.834} C_VEL
LIN {X 0,Y 209.649,Z 355.846,A -85,B 0,C 180,E1 -21663.63,E2 -21663.63} C_VEL
LIN {X 0,Y 208.348,Z 360.212,A -85,B 0,C 180,E1 -21664.689,E2 -21664.689} C_VEL
LIN {X 0,Y 206.44,Z 364.302,A -85,B 0,C 180,E1 -21665.75,E2 -21665.75} C_VEL
LIN {X 0,Y 201.701,Z 370.601,A -85,B 0,C 180,E1 -21667.453,E2 -21667.453} C_VEL
LIN {X 0,Y 197.044,Z 376.292,A -85,B 0,C 180,E1 -21669.369,E2 -21669.369} C_VEL
LIN {X 0,Y 195.311,Z 379.426,A -85,B 0,C 180,E1 -21670.743,E2 -21670.743} C_VEL
LIN {X 0,Y 193.034,Z 385.602,A -85,B 0,C 180,E1 -21674.154,E2 -21674.154} C_VEL
LIN {X 0,Y 191.642,Z 389.931,A -85,B 0,C 180,E1 -21677.289,E2 -21677.289} C_VEL
LIN {X 0,Y 190.995,Z 392.302,A -85,B 0,C 180,E1 -21679.398,E2 -21679.398} C_VEL
LIN {X 0,Y 190.528,Z 394.105,A -85,B 0,C 180,E1 -21681.515,E2 -21681.515} C_VEL
LIN {X 0,Y 190.166,Z 396.561,A -85,B 0,C 180,E1 -21685.761,E2 -21685.761} C_VEL
LIN {X 0,Y 190.152,Z 397.155,A -85,B 0,C 180,E1 -21687.882,E2 -21687.882} C_VEL
LIN {X 0,Y 190.244,Z 397.313,A -85,B 0,C 180,E1 -21690,E2 -21690} C_VEL
LIN {X 0,Y 190.12,Z 396.76,A -85,B 0,C 180,E1 -21693.529,E2 -21693.529} C_VEL
LIN {X 0,Y 190.231,Z 395.497,A -85,B 0,C 180,E1 -21696.363,E2 -21696.363} C_VEL
LIN {X 0,Y 190.502,Z 394.104,A -85,B 0,C 180,E1 -21698.486,E2 -21698.486} C_VEL
LIN {X 0,Y 191.279,Z 391.149,A -85,B 0,C 180,E1 -21701.659,E2 -21701.659} C_VEL
LIN {X 0,Y 192.462,Z 387.156,A -85,B 0,C 180,E1 -21704.81,E2 -21704.81} C_VEL
LIN {X 0,Y 194.343,Z 382.027,A -85,B 0,C 180,E1 -21707.901,E2 -21707.901} C_VEL
LIN {X 0,Y 196.22,Z 376.765,A -85,B 0,C 180,E1 -21710.439,E2 -21710.439} C_VEL
LIN {X 0,Y 198.131,Z 371.509,A -85,B 0,C 180,E1 -21712.542,E2 -21712.542} C_VEL
LIN {X 0,Y 200.419,Z 364.498,A -85,B 0,C 180,E1 -21714.885,E2 -21714.885} C_VEL
LIN {X 0,Y 202.701,Z 357.573,A -85,B 0,C 180,E1 -21716.79,E2 -21716.79} C_VEL
LIN {X 0,Y 205.246,Z 349.398,A -85,B 0,C 180,E1 -21718.645,E2 -21718.645} C_VEL
LIN {X 0,Y 207.648,Z 340.891,A -85,B 0,C 180,E1 -21720.228,E2 -21720.228} C_VEL
LIN {X 0,Y 209.907,Z 332.181,A -85,B 0,C 180,E1 -21721.543,E2 -21721.543} C_VEL
LIN {X 0,Y 212.016,Z 322.427,A -85,B 0,C 180,E1 -21722.733,E2 -21722.733} C_VEL
LIN {X 0,Y 213.61,Z 313.635,A -85,B 0,C 180,E1 -21723.583,E2 -21723.583} C_VEL
LIN {X 0,Y 215.153,Z 303.318,A -85,B 0,C 180,E1 -21724.328,E2 -21724.328} C_VEL
LIN {X 0,Y 216.137,Z 293.274,A -85,B 0,C 180,E1 -21724.855,E2 -21724.855} C_VEL
LIN {X 0,Y 217.737,Z 262.26,A -85,B 0,C 180,E1 -21725.869,E2 -21725.869} C_VEL
LIN {X 0,Y 218.404,Z 247.431,A -85,B 0,C 180,E1 -21726.333,E2 -21726.333} C_VEL
LIN {X 0,Y 215.726,Z 230.653,A -85,B 0,C 180,E1 -21727.539,E2 -21727.539} C_VEL
LIN {X 0,Y 209.91,Z 216.821,A -85,B 0,C 180,E1 -21729.356,E2 -21729.356} C_VEL
LIN {X 0,Y 203.789,Z 204.179,A -85,B 0,C 180,E1 -21731.349,E2 -21731.349} C_VEL
LIN {X 0,Y 198.449,Z 194.701,A -85,B 0,C 180,E1 -21733.169,E2 -21733.169} C_VEL
LIN {X 0,Y 195.509,Z 189.704,A -85,B 0,C 180,E1 -21734.227,E2 -21734.227} C_VEL
LIN {X 0,Y 193.567,Z 185.897,A -85,B 0,C 180,E1 -21735.11,E2 -21735.11} C_VEL
LIN {X 0,Y 192.54,Z 182.071,A -85,B 0,C 180,E1 -21738.222,E2 -21738.222} C_VEL
LIN {X 0,Y 192.588,Z 181.986,A -85,B 0,C 180,E1 -21743.4,E2 -21743.4} C_VEL
LIN {X 0,Y 192.611,Z 181.967,A -85,B 0,C 180,E1 -21747.057,E2 -21747.057} C_VEL
LIN {X 0,Y 192.665,Z 181.954,A -85,B 0,C 180,E1 -21751.691,E2 -21751.691} C_VEL
LIN {X 0,Y 192.706,Z 181.976,A -85,B 0,C 180,E1 -21756.347,E2 -21756.347} C_VEL
LIN {X 0,Y 192.732,Z 181.929,A -85,B 0,C 180,E1 -21761.457,E2 -21761.457} C_VEL
LIN {X 0,Y 192.764,Z 181.969,A -85,B 0,C 180,E1 -21765.213,E2 -21765.213} C_VEL
LIN {X 0,Y 192.945,Z 181.901,A -85,B 0,C 180,E1 -21769.565,E2 -21769.565} C_VEL
LIN {X 0,Y 192.985,Z 181.933,A -85,B 0,C 180,E1 -21773.727,E2 -21773.727} C_VEL
LIN {X 0,Y 193.262,Z 181.877,A -85,B 0,C 180,E1 -21777.915,E2 -21777.915} C_VEL
LIN {X 0,Y 193.439,Z 181.836,A -85,B 0,C 180,E1 -21779.999,E2 -21779.999} C_VEL
LIN {X 0,Y 192.977,Z 181.943,A -85,B 0,C 180,E1 -21784.176,E2 -21784.176} C_VEL
LIN {X 0,Y 193.06,Z 181.894,A -85,B 0,C 180,E1 -21788.372,E2 -21788.372} C_VEL
LIN {X 0,Y 192.851,Z 181.939,A -85,B 0,C 180,E1 -21792.629,E2 -21792.629} C_VEL
LIN {X 0,Y 192.756,Z 181.945,A -85,B 0,C 180,E1 -21796.958,E2 -21796.958} C_VEL
LIN {X 0,Y 192.634,Z 181.964,A -85,B 0,C 180,E1 -21801.396,E2 -21801.396} C_VEL
LIN {X 0,Y 192.662,Z 181.981,A -85,B 0,C 180,E1 -21804.224,E2 -21804.224} C_VEL
LIN {X 0,Y 192.647,Z 181.96,A -85,B 0,C 180,E1 -21808.891,E2 -21808.891} C_VEL
LIN {X 0,Y 192.597,Z 181.971,A -85,B 0,C 180,E1 -21813.185,E2 -21813.185} C_VEL
LIN {X 0,Y 192.571,Z 181.994,A -85,B 0,C 180,E1 -21818.346,E2 -21818.346} C_VEL
LIN {X 0,Y 192.511,Z 182.003,A -85,B 0,C 180,E1 -21823.103,E2 -21823.103} C_VEL
LIN {X 0,Y 192.584,Z 182.263,A -85,B 0,C 180,E1 -21824.642,E2 -21824.642} C_VEL
LIN {X 0,Y 192.895,Z 183.403,A -85,B 0,C 180,E1 -21825.052,E2 -21825.052} C_VEL
LIN {X 0,Y 194.497,Z 186.091,A -85,B 0,C 180,E1 -21825.681,E2 -21825.681} C_VEL
LIN {X 0,Y 195.872,Z 187.655,A -85,B 0,C 180,E1 -21826.153,E2 -21826.153} C_VEL
LIN {X 0,Y 197.956,Z 190.791,A -85,B 0,C 180,E1 -21826.887,E2 -21826.887} C_VEL
LIN {X 0,Y 203.577,Z 199.281,A -85,B 0,C 180,E1 -21828.753,E2 -21828.753} C_VEL
LIN {X 0,Y 210.683,Z 211.16,A -85,B 0,C 180,E1 -21830.951,E2 -21830.951} C_VEL
LIN {X 0,Y 218.645,Z 226.643,A -85,B 0,C 180,E1 -21833.261,E2 -21833.261} C_VEL
LIN {X 0,Y 225.879,Z 241.544,A -85,B 0,C 180,E1 -21835.197,E2 -21835.197} C_VEL
LIN {X 0,Y 234.469,Z 255.413,A -85,B 0,C 180,E1 -21837.151,E2 -21837.151} C_VEL
LIN {X 0,Y 242.462,Z 266.178,A -85,B 0,C 180,E1 -21838.738,E2 -21838.738} C_VEL
LIN {X 0,Y 254.128,Z 279.577,A -85,B 0,C 180,E1 -21840.792,E2 -21840.792} C_VEL
LIN {X 0,Y 265.228,Z 290.848,A -85,B 0,C 180,E1 -21842.685,E2 -21842.685} C_VEL
LIN {X 0,Y 276.274,Z 300.759,A -85,B 0,C 180,E1 -21844.56,E2 -21844.56} C_VEL
LIN {X 0,Y 290.367,Z 312.016,A -85,B 0,C 180,E1 -21846.887,E2 -21846.887} C_VEL
LIN {X 0,Y 300.18,Z 319.525,A -85,B 0,C 180,E1 -21848.534,E2 -21848.534} C_VEL
LIN {X 0,Y 307.937,Z 325.193,A -85,B 0,C 180,E1 -21849.981,E2 -21849.981} C_VEL
LIN {X 0,Y 314.999,Z 330.316,A -85,B 0,C 180,E1 -21851.482,E2 -21851.482} C_VEL
LIN {X 0,Y 321.422,Z 334.728,A -85,B 0,C 180,E1 -21852.992,E2 -21852.992} C_VEL
LIN {X 0,Y 327.802,Z 339.364,A -85,B 0,C 180,E1 -21854.747,E2 -21854.747} C_VEL
LIN {X 0,Y 334.13,Z 343.194,A -85,B 0,C 180,E1 -21856.622,E2 -21856.622} C_VEL
LIN {X 0,Y 338.056,Z 345.795,A -85,B 0,C 180,E1 -21858.001,E2 -21858.001} C_VEL
LIN {X 0,Y 342.61,Z 349.004,A -85,B 0,C 180,E1 -21859.937,E2 -21859.937} C_VEL
LIN {X 0,Y 347.431,Z 351.907,A -85,B 0,C 180,E1 -21862.385,E2 -21862.385} C_VEL
LIN {X 0,Y 350.395,Z 353.322,A -85,B 0,C 180,E1 -21864.244,E2 -21864.244} C_VEL
LIN {X 0,Y 352.331,Z 354.1,A -85,B 0,C 180,E1 -21865.823,E2 -21865.823} C_VEL
LIN {X 0,Y 353.098,Z 354.347,A -85,B 0,C 180,E1 -21866.577,E2 -21866.577} C_VEL
LIN {X 0,Y 353.872,Z 354.705,A -85,B 0,C 180,E1 -21867.724,E2 -21867.724} C_VEL
LIN {X 0,Y 354.286,Z 354.956,A -85,B 0,C 180,E1 -21868.863,E2 -21868.863} C_VEL
LIN {X 0,Y 354.529,Z 354.92,A -85,B 0,C 180,E1 -21870,E2 -21870} C_VEL
LIN {X 0,Y 354.29,Z 354.936,A -85,B 0,C 180,E1 -21871.137,E2 -21871.137} C_VEL
LIN {X 0,Y 353.873,Z 354.677,A -85,B 0,C 180,E1 -21872.276,E2 -21872.276} C_VEL
LIN {X 0,Y 352.339,Z 354.102,A -85,B 0,C 180,E1 -21874.196,E2 -21874.196} C_VEL
LIN {X 0,Y 350.367,Z 353.305,A -85,B 0,C 180,E1 -21875.756,E2 -21875.756} C_VEL
LIN {X 0,Y 347.436,Z 351.93,A -85,B 0,C 180,E1 -21877.621,E2 -21877.621} C_VEL
LIN {X 0,Y 342.614,Z 348.984,A -85,B 0,C 180,E1 -21880.067,E2 -21880.067} C_VEL
LIN {X 0,Y 338.025,Z 345.761,A -85,B 0,C 180,E1 -21882,E2 -21882} C_VEL
LIN {X 0,Y 334.116,Z 343.229,A -85,B 0,C 180,E1 -21883.378,E2 -21883.378} C_VEL
LIN {X 0,Y 327.802,Z 339.351,A -85,B 0,C 180,E1 -21885.253,E2 -21885.253} C_VEL
LIN {X 0,Y 321.389,Z 334.736,A -85,B 0,C 180,E1 -21887.006,E2 -21887.006} C_VEL
LIN {X 0,Y 314.989,Z 330.328,A -85,B 0,C 180,E1 -21888.513,E2 -21888.513} C_VEL
LIN {X 0,Y 307.025,Z 324.52,A -85,B 0,C 180,E1 -21890.199,E2 -21890.199} C_VEL
LIN {X 0,Y 298.791,Z 318.528,A -85,B 0,C 180,E1 -21891.708,E2 -21891.708} C_VEL
LIN {X 0,Y 287.539,Z 309.894,A -85,B 0,C 180,E1 -21893.572,E2 -21893.572} C_VEL
LIN {X 0,Y 273.475,Z 298.39,A -85,B 0,C 180,E1 -21895.915,E2 -21895.915} C_VEL
LIN {X 0,Y 261.035,Z 286.699,A -85,B 0,C 180,E1 -21898.046,E2 -21898.046} C_VEL
LIN {X 0,Y 249.896,Z 274.907,A -85,B 0,C 180,E1 -21899.941,E2 -21899.941} C_VEL
LIN {X 0,Y 238.274,Z 260.818,A -85,B 0,C 180,E1 -21902.067,E2 -21902.067} C_VEL
LIN {X 0,Y 229.169,Z 247.149,A -85,B 0,C 180,E1 -21904.021,E2 -21904.021} C_VEL
LIN {X 0,Y 221.957,Z 233.9,A -85,B 0,C 180,E1 -21905.814,E2 -21905.814} C_VEL
LIN {X 0,Y 214.999,Z 219.38,A -85,B 0,C 180,E1 -21907.774,E2 -21907.774} C_VEL
LIN {X 0,Y 207.618,Z 205.762,A -85,B 0,C 180,E1 -21909.982,E2 -21909.982} C_VEL
LIN {X 0,Y 200.303,Z 194.299,A -85,B 0,C 180,E1 -21912.316,E2 -21912.316} C_VEL
LIN {X 0,Y 197.662,Z 190.483,A -85,B 0,C 180,E1 -21913.208,E2 -21913.208} C_VEL
LIN {X 0,Y 195.24,Z 186.772,A -85,B 0,C 180,E1 -21914.071,E2 -21914.071} C_VEL
LIN {X 0,Y 193.303,Z 184.406,A -85,B 0,C 180,E1 -21914.755,E2 -21914.755} C_VEL
LIN {X 0,Y 192.621,Z 182.456,A -85,B 0,C 180,E1 -21915.244,E2 -21915.244} C_VEL
LIN {X 0,Y 192.511,Z 182,A -85,B 0,C 180,E1 -21916.083,E2 -21916.083} C_VEL
LIN {X 0,Y 192.537,Z 181.98,A -85,B 0,C 180,E1 -21920.044,E2 -21920.044} C_VEL
LIN {X 0,Y 192.578,Z 181.973,A -85,B 0,C 180,E1 -21924.276,E2 -21924.276} C_VEL
LIN {X 0,Y 192.605,Z 181.995,A -85,B 0,C 180,E1 -21929.281,E2 -21929.281} C_VEL
LIN {X 0,Y 192.662,Z 181.953,A -85,B 0,C 180,E1 -21931.693,E2 -21931.693} C_VEL
LIN {X 0,Y 192.703,Z 181.981,A -85,B 0,C 180,E1 -21936.35,E2 -21936.35} C_VEL
LIN {X 0,Y 192.73,Z 181.933,A -85,B 0,C 180,E1 -21941.459,E2 -21941.459} C_VEL
LIN {X 0,Y 192.77,Z 181.973,A -85,B 0,C 180,E1 -21945.215,E2 -21945.215} C_VEL
LIN {X 0,Y 192.979,Z 181.897,A -85,B 0,C 180,E1 -21949.51,E2 -21949.51} C_VEL
LIN {X 0,Y 193.06,Z 181.894,A -85,B 0,C 180,E1 -21951.628,E2 -21951.628} C_VEL
LIN {X 0,Y 193.263,Z 181.872,A -85,B 0,C 180,E1 -21957.917,E2 -21957.917} C_VEL
LIN {X 0,Y 193.439,Z 181.836,A -85,B 0,C 180,E1 -21960.001,E2 -21960.001} C_VEL
LIN {X 0,Y 192.973,Z 181.946,A -85,B 0,C 180,E1 -21964.178,E2 -21964.178} C_VEL
LIN {X 0,Y 193.036,Z 181.893,A -85,B 0,C 180,E1 -21968.375,E2 -21968.375} C_VEL
LIN {X 0,Y 192.802,Z 181.948,A -85,B 0,C 180,E1 -21972.635,E2 -21972.635} C_VEL
LIN {X 0,Y 192.758,Z 181.937,A -85,B 0,C 180,E1 -21976.96,E2 -21976.96} C_VEL
LIN {X 0,Y 192.637,Z 181.967,A -85,B 0,C 180,E1 -21981.398,E2 -21981.398} C_VEL
LIN {X 0,Y 192.665,Z 181.973,A -85,B 0,C 180,E1 -21984.226,E2 -21984.226} C_VEL
LIN {X 0,Y 192.651,Z 181.963,A -85,B 0,C 180,E1 -21988.893,E2 -21988.893} C_VEL
LIN {X 0,Y 192.6,Z 181.967,A -85,B 0,C 180,E1 -21993.187,E2 -21993.187} C_VEL
LIN {X 0,Y 192.553,Z 181.99,A -85,B 0,C 180,E1 -21998.353,E2 -21998.353} C_VEL
LIN {X 0,Y 192.57,Z 182.169,A -85,B 0,C 180,E1 -22001.916,E2 -22001.916} C_VEL
LIN {X 0,Y 193.544,Z 185.936,A -85,B 0,C 180,E1 -22004.897,E2 -22004.897} C_VEL
LIN {X 0,Y 195.803,Z 190.171,A -85,B 0,C 180,E1 -22005.88,E2 -22005.88} C_VEL
LIN {X 0,Y 200.568,Z 198.409,A -85,B 0,C 180,E1 -22007.568,E2 -22007.568} C_VEL
LIN {X 0,Y 204.703,Z 205.957,A -85,B 0,C 180,E1 -22008.955,E2 -22008.955} C_VEL
LIN {X 0,Y 210.49,Z 218.131,A -85,B 0,C 180,E1 -22010.829,E2 -22010.829} C_VEL
LIN {X 0,Y 215.86,Z 231.021,A -85,B 0,C 180,E1 -22012.503,E2 -22012.503} C_VEL
LIN {X 0,Y 218.463,Z 248.206,A -85,B 0,C 180,E1 -22013.709,E2 -22013.709} C_VEL
LIN {X 0,Y 216.31,Z 292.31,A -85,B 0,C 180,E1 -22015.119,E2 -22015.119} C_VEL
LIN {X 0,Y 215.187,Z 303.306,A -85,B 0,C 180,E1 -22015.677,E2 -22015.677} C_VEL
LIN {X 0,Y 213.643,Z 313.637,A -85,B 0,C 180,E1 -22016.423,E2 -22016.423} C_VEL
LIN {X 0,Y 211.648,Z 324.441,A -85,B 0,C 180,E1 -22017.485,E2 -22017.485} C_VEL
LIN {X 0,Y 208.822,Z 336.841,A -85,B 0,C 180,E1 -22019.12,E2 -22019.12} C_VEL
LIN {X 0,Y 205.934,Z 347.131,A -85,B 0,C 180,E1 -22020.902,E2 -22020.902} C_VEL
LIN {X 0,Y 203.306,Z 355.655,A -85,B 0,C 180,E1 -22022.74,E2 -22022.74} C_VEL
LIN {X 0,Y 200.965,Z 362.871,A -85,B 0,C 180,E1 -22024.634,E2 -22024.634} C_VEL
LIN {X 0,Y 198.857,Z 369.071,A -85,B 0,C 180,E1 -22026.572,E2 -22026.572} C_VEL
LIN {X 0,Y 196.689,Z 375.611,A -85,B 0,C 180,E1 -22029.065,E2 -22029.065} C_VEL
LIN {X 0,Y 195.311,Z 379.426,A -85,B 0,C 180,E1 -22030.743,E2 -22030.743} C_VEL
LIN {X 0,Y 193.645,Z 382.312,A -85,B 0,C 180,E1 -22032.183,E2 -22032.183} C_VEL
LIN {X 0,Y 191.164,Z 384.977,A -85,B 0,C 180,E1 -22033.595,E2 -22033.595} C_VEL
LIN {X 0,Y 185.269,Z 390.056,A -85,B 0,C 180,E1 -22037.097,E2 -22037.097} C_VEL
LIN {X 0,Y 184.033,Z 391.9,A -85,B 0,C 180,E1 -22038.79,E2 -22038.79} C_VEL
LIN {X 0,Y 183.499,Z 393.913,A -85,B 0,C 180,E1 -22041.188,E2 -22041.188} C_VEL
LIN {X 0,Y 183.08,Z 396.37,A -85,B 0,C 180,E1 -22045.597,E2 -22045.597} C_VEL
LIN {X 0,Y 183.05,Z 396.963,A -85,B 0,C 180,E1 -22047.8,E2 -22047.8} C_VEL
LIN {X 0,Y 183.15,Z 397.121,A -85,B 0,C 180,E1 -22050,E2 -22050} C_VEL
LIN {X 0,Y 183.035,Z 396.667,A -85,B 0,C 180,E1 -22053.301,E2 -22053.301} C_VEL
LIN {X 0,Y 183.149,Z 395.304,A -85,B 0,C 180,E1 -22056.61,E2 -22056.61} C_VEL
LIN {X 0,Y 183.453,Z 393.912,A -85,B 0,C 180,E1 -22058.815,E2 -22058.815} C_VEL
LIN {X 0,Y 184.312,Z 390.957,A -85,B 0,C 180,E1 -22062.106,E2 -22062.106} C_VEL
LIN {X 0,Y 185.571,Z 386.963,A -85,B 0,C 180,E1 -22065.373,E2 -22065.373} C_VEL
LIN {X 0,Y 187.578,Z 381.835,A -85,B 0,C 180,E1 -22068.57,E2 -22068.57} C_VEL
LIN {X 0,Y 189.579,Z 376.574,A -85,B 0,C 180,E1 -22071.189,E2 -22071.189} C_VEL
LIN {X 0,Y 191.764,Z 370.635,A -85,B 0,C 180,E1 -22073.617,E2 -22073.617} C_VEL
LIN {X 0,Y 193.966,Z 364.305,A -85,B 0,C 180,E1 -22075.772,E2 -22075.772} C_VEL
LIN {X 0,Y 196.386,Z 357.381,A -85,B 0,C 180,E1 -22077.725,E2 -22077.725} C_VEL
LIN {X 0,Y 199.02,Z 349.206,A -85,B 0,C 180,E1 -22079.629,E2 -22079.629} C_VEL
LIN {X 0,Y 201.543,Z 340.699,A -85,B 0,C 180,E1 -22081.245,E2 -22081.245} C_VEL
LIN {X 0,Y 203.89,Z 331.99,A -85,B 0,C 180,E1 -22082.587,E2 -22082.587} C_VEL
LIN {X 0,Y 206.078,Z 322.235,A -85,B 0,C 180,E1 -22083.801,E2 -22083.801} C_VEL
LIN {X 0,Y 207.741,Z 313.444,A -85,B 0,C 180,E1 -22084.665,E2 -22084.665} C_VEL
LIN {X 0,Y 209.404,Z 302.713,A -85,B 0,C 180,E1 -22085.444,E2 -22085.444} C_VEL
LIN {X 0,Y 210.357,Z 292.877,A -85,B 0,C 180,E1 -22085.971,E2 -22085.971} C_VEL
LIN {X 0,Y 212.105,Z 260.567,A -85,B 0,C 180,E1 -22087.039,E2 -22087.039} C_VEL
LIN {X 0,Y 212.634,Z 247.947,A -85,B 0,C 180,E1 -22087.455,E2 -22087.455} C_VEL
LIN {X 0,Y 210.203,Z 233.143,A -85,B 0,C 180,E1 -22088.591,E2 -22088.591} C_VEL
LIN {X 0,Y 204.33,Z 219.108,A -85,B 0,C 180,E1 -22090.539,E2 -22090.539} C_VEL
LIN {X 0,Y 198.399,Z 206.895,A -85,B 0,C 180,E1 -22092.594,E2 -22092.594} C_VEL
LIN {X 0,Y 191.843,Z 195.222,A -85,B 0,C 180,E1 -22095.009,E2 -22095.009} C_VEL
LIN {X 0,Y 188.914,Z 190.358,A -85,B 0,C 180,E1 -22096.159,E2 -22096.159} C_VEL
LIN {X 0,Y 186.375,Z 186.199,A -85,B 0,C 180,E1 -22097.252,E2 -22097.252} C_VEL
LIN {X 0,Y 186.018,Z 185.09,A -85,B 0,C 180,E1 -22097.772,E2 -22097.772} C_VEL
LIN {X 0,Y 185.473,Z 182.885,A -85,B 0,C 180,E1 -22099.895,E2 -22099.895} C_VEL
LIN {X 0,Y 185.509,Z 182.878,A -85,B 0,C 180,E1 -22102.709,E2 -22102.709} C_VEL
LIN {X 0,Y 185.547,Z 182.857,A -85,B 0,C 180,E1 -22107.974,E2 -22107.974} C_VEL
LIN {X 0,Y 185.583,Z 182.85,A -85,B 0,C 180,E1 -22110.575,E2 -22110.575} C_VEL
LIN {X 0,Y 185.588,Z 182.846,A -85,B 0,C 180,E1 -22115.381,E2 -22115.381} C_VEL
LIN {X 0,Y 185.607,Z 182.821,A -85,B 0,C 180,E1 -22120.074,E2 -22120.074} C_VEL
LIN {X 0,Y 185.695,Z 182.842,A -85,B 0,C 180,E1 -22124.636,E2 -22124.636} C_VEL
LIN {X 0,Y 185.888,Z 182.779,A -85,B 0,C 180,E1 -22129.417,E2 -22129.417} C_VEL
LIN {X 0,Y 185.947,Z 182.803,A -85,B 0,C 180,E1 -22133.488,E2 -22133.488} C_VEL
LIN {X 0,Y 186.206,Z 182.755,A -85,B 0,C 180,E1 -22137.836,E2 -22137.836} C_VEL
LIN {X 0,Y 186.403,Z 182.712,A -85,B 0,C 180,E1 -22139.999,E2 -22139.999} C_VEL
LIN {X 0,Y 185.925,Z 182.822,A -85,B 0,C 180,E1 -22144.335,E2 -22144.335} C_VEL
LIN {X 0,Y 186.007,Z 182.768,A -85,B 0,C 180,E1 -22148.691,E2 -22148.691} C_VEL
LIN {X 0,Y 185.763,Z 182.831,A -85,B 0,C 180,E1 -22153.119,E2 -22153.119} C_VEL
LIN {X 0,Y 185.688,Z 182.815,A -85,B 0,C 180,E1 -22157.624,E2 -22157.624} C_VEL
LIN {X 0,Y 185.594,Z 182.856,A -85,B 0,C 180,E1 -22162.25,E2 -22162.25} C_VEL
LIN {X 0,Y 185.56,Z 182.833,A -85,B 0,C 180,E1 -22167.031,E2 -22167.031} C_VEL
LIN {X 0,Y 185.576,Z 182.848,A -85,B 0,C 180,E1 -22169.492,E2 -22169.492} C_VEL
LIN {X 0,Y 185.507,Z 182.847,A -85,B 0,C 180,E1 -22174.629,E2 -22174.629} C_VEL
LIN {X 0,Y 185.541,Z 182.871,A -85,B 0,C 180,E1 -22177.303,E2 -22177.303} C_VEL
LIN {X 0,Y 185.455,Z 182.973,A -85,B 0,C 180,E1 -22182.231,E2 -22182.231} C_VEL
LIN {X 0,Y 185.688,Z 183.982,A -85,B 0,C 180,E1 -22182.785,E2 -22182.785} C_VEL
LIN {X 0,Y 187.298,Z 186.826,A -85,B 0,C 180,E1 -22183.514,E2 -22183.514} C_VEL
LIN {X 0,Y 188.835,Z 188.369,A -85,B 0,C 180,E1 -22184.089,E2 -22184.089} C_VEL
LIN {X 0,Y 190.882,Z 191.609,A -85,B 0,C 180,E1 -22184.894,E2 -22184.894} C_VEL
LIN {X 0,Y 192.206,Z 193.407,A -85,B 0,C 180,E1 -22185.384,E2 -22185.384} C_VEL
LIN {X 0,Y 197.875,Z 201.848,A -85,B 0,C 180,E1 -22187.403,E2 -22187.403} C_VEL
LIN {X 0,Y 205.232,Z 214.048,A -85,B 0,C 180,E1 -22189.827,E2 -22189.827} C_VEL
LIN {X 0,Y 213.074,Z 229.359,A -85,B 0,C 180,E1 -22192.24,E2 -22192.24} C_VEL
LIN {X 0,Y 221.263,Z 246.355,A -85,B 0,C 180,E1 -22194.544,E2 -22194.544} C_VEL
LIN {X 0,Y 229.961,Z 260.433,A -85,B 0,C 180,E1 -22196.602,E2 -22196.602} C_VEL
LIN {X 0,Y 237.788,Z 271.069,A -85,B 0,C 180,E1 -22198.217,E2 -22198.217} C_VEL
LIN {X 0,Y 248.144,Z 283.148,A -85,B 0,C 180,E1 -22200.152,E2 -22200.152} C_VEL
LIN {X 0,Y 259.309,Z 294.901,A -85,B 0,C 180,E1 -22202.259,E2 -22202.259} C_VEL
LIN {X 0,Y 272.194,Z 306.586,A -85,B 0,C 180,E1 -22204.646,E2 -22204.646} C_VEL
LIN {X 0,Y 286.085,Z 317.594,A -85,B 0,C 180,E1 -22207.104,E2 -22207.104} C_VEL
LIN {X 0,Y 298.882,Z 327.145,A -85,B 0,C 180,E1 -22209.347,E2 -22209.347} C_VEL
LIN {X 0,Y 305.408,Z 332.038,A -85,B 0,C 180,E1 -22210.643,E2 -22210.643} C_VEL
LIN {X 0,Y 313.311,Z 337.519,A -85,B 0,C 180,E1 -22212.37,E2 -22212.37} C_VEL
LIN {X 0,Y 318.531,Z 341.303,A -85,B 0,C 180,E1 -22213.689,E2 -22213.689} C_VEL
LIN {X 0,Y 325.221,Z 345.882,A -85,B 0,C 180,E1 -22215.562,E2 -22215.562} C_VEL
LIN {X 0,Y 331.231,Z 349.467,A -85,B 0,C 180,E1 -22217.423,E2 -22217.423} C_VEL
LIN {X 0,Y 336.078,Z 352.937,A -85,B 0,C 180,E1 -22219.371,E2 -22219.371} C_VEL
LIN {X 0,Y 338.427,Z 354.534,A -85,B 0,C 180,E1 -22220.437,E2 -22220.437} C_VEL
LIN {X 0,Y 340.952,Z 356.092,A -85,B 0,C 180,E1 -22221.704,E2 -22221.704} C_VEL
LIN {X 0,Y 343.227,Z 357.278,A -85,B 0,C 180,E1 -22222.943,E2 -22222.943} C_VEL
LIN {X 0,Y 345.849,Z 358.517,A -85,B 0,C 180,E1 -22224.694,E2 -22224.694} C_VEL
LIN {X 0,Y 347.953,Z 359.289,A -85,B 0,C 180,E1 -22226.526,E2 -22226.526} C_VEL
LIN {X 0,Y 348.771,Z 359.649,A -85,B 0,C 180,E1 -22227.69,E2 -22227.69} C_VEL
LIN {X 0,Y 349.197,Z 359.912,A -85,B 0,C 180,E1 -22228.847,E2 -22228.847} C_VEL
LIN {X 0,Y 349.469,Z 359.876,A -85,B 0,C 180,E1 -22230,E2 -22230} C_VEL
LIN {X 0,Y 349.212,Z 359.884,A -85,B 0,C 180,E1 -22231.153,E2 -22231.153} C_VEL
LIN {X 0,Y 348.771,Z 359.624,A -85,B 0,C 180,E1 -22232.31,E2 -22232.31} C_VEL
LIN {X 0,Y 347.952,Z 359.257,A -85,B 0,C 180,E1 -22233.474,E2 -22233.474} C_VEL
LIN {X 0,Y 345.856,Z 358.533,A -85,B 0,C 180,E1 -22235.318,E2 -22235.318} C_VEL
LIN {X 0,Y 343.185,Z 357.279,A -85,B 0,C 180,E1 -22237.058,E2 -22237.058} C_VEL
LIN {X 0,Y 340.925,Z 356.036,A -85,B 0,C 180,E1 -22238.318,E2 -22238.318} C_VEL
LIN {X 0,Y 338.449,Z 354.49,A -85,B 0,C 180,E1 -22239.562,E2 -22239.562} C_VEL
LIN {X 0,Y 334.446,Z 351.801,A -85,B 0,C 180,E1 -22241.325,E2 -22241.325} C_VEL
LIN {X 0,Y 331.228,Z 349.521,A -85,B 0,C 180,E1 -22242.575,E2 -22242.575} C_VEL
LIN {X 0,Y 325.23,Z 345.872,A -85,B 0,C 180,E1 -22244.437,E2 -22244.437} C_VEL
LIN {X 0,Y 318.53,Z 341.293,A -85,B 0,C 180,E1 -22246.311,E2 -22246.311} C_VEL
LIN {X 0,Y 313.278,Z 337.537,A -85,B 0,C 180,E1 -22247.637,E2 -22247.637} C_VEL
LIN {X 0,Y 305.403,Z 332.056,A -85,B 0,C 180,E1 -22249.355,E2 -22249.355} C_VEL
LIN {X 0,Y 297.243,Z 325.969,A -85,B 0,C 180,E1 -22250.944,E2 -22250.944} C_VEL
LIN {X 0,Y 283.189,Z 315.441,A -85,B 0,C 180,E1 -22253.395,E2 -22253.395} C_VEL
LIN {X 0,Y 270.678,Z 305.282,A -85,B 0,C 180,E1 -22255.635,E2 -22255.635} C_VEL
LIN {X 0,Y 258.283,Z 293.867,A -85,B 0,C 180,E1 -22257.936,E2 -22257.936} C_VEL
LIN {X 0,Y 247.285,Z 282.188,A -85,B 0,C 180,E1 -22260.011,E2 -22260.011} C_VEL
LIN {X 0,Y 235.775,Z 268.591,A -85,B 0,C 180,E1 -22262.176,E2 -22262.176} C_VEL
LIN {X 0,Y 225.309,Z 253.275,A -85,B 0,C 180,E1 -22264.459,E2 -22264.459} C_VEL
LIN {X 0,Y 218.136,Z 240.297,A -85,B 0,C 180,E1 -22266.29,E2 -22266.29} C_VEL
LIN {X 0,Y 210.296,Z 223.736,A -85,B 0,C 180,E1 -22268.593,E2 -22268.593} C_VEL
LIN {X 0,Y 203.119,Z 210.302,A -85,B 0,C 180,E1 -22270.853,E2 -22270.853} C_VEL
LIN {X 0,Y 195.852,Z 198.733,A -85,B 0,C 180,E1 -22273.301,E2 -22273.301} C_VEL
LIN {X 0,Y 191.171,Z 191.925,A -85,B 0,C 180,E1 -22275.002,E2 -22275.002} C_VEL
LIN {X 0,Y 188.927,Z 188.556,A -85,B 0,C 180,E1 -22275.872,E2 -22275.872} C_VEL
LIN {X 0,Y 187.921,Z 187.389,A -85,B 0,C 180,E1 -22276.254,E2 -22276.254} C_VEL
LIN {X 0,Y 186.219,Z 185.268,A -85,B 0,C 180,E1 -22276.925,E2 -22276.925} C_VEL
LIN {X 0,Y 185.513,Z 183.312,A -85,B 0,C 180,E1 -22277.476,E2 -22277.476} C_VEL
LIN {X 0,Y 185.463,Z 182.888,A -85,B 0,C 180,E1 -22278.233,E2 -22278.233} C_VEL
LIN {X 0,Y 185.541,Z 182.871,A -85,B 0,C 180,E1 -22282.697,E2 -22282.697} C_VEL
LIN {X 0,Y 185.542,Z 182.864,A -85,B 0,C 180,E1 -22287.976,E2 -22287.976} C_VEL
LIN {X 0,Y 185.579,Z 182.846,A -85,B 0,C 180,E1 -22290.577,E2 -22290.577} C_VEL
LIN {X 0,Y 185.585,Z 182.855,A -85,B 0,C 180,E1 -22295.384,E2 -22295.384} C_VEL
LIN {X 0,Y 185.605,Z 182.821,A -85,B 0,C 180,E1 -22300.076,E2 -22300.076} C_VEL
LIN {X 0,Y 185.723,Z 182.847,A -85,B 0,C 180,E1 -22304.641,E2 -22304.641} C_VEL
LIN {X 0,Y 185.922,Z 182.776,A -85,B 0,C 180,E1 -22309.36,E2 -22309.36} C_VEL
LIN {X 0,Y 185.96,Z 182.807,A -85,B 0,C 180,E1 -22313.491,E2 -22313.491} C_VEL
LIN {X 0,Y 186.207,Z 182.75,A -85,B 0,C 180,E1 -22317.838,E2 -22317.838} C_VEL
LIN {X 0,Y 186.403,Z 182.712,A -85,B 0,C 180,E1 -22320.001,E2 -22320.001} C_VEL
LIN {X 0,Y 185.92,Z 182.826,A -85,B 0,C 180,E1 -22324.337,E2 -22324.337} C_VEL
LIN {X 0,Y 185.982,Z 182.768,A -85,B 0,C 180,E1 -22328.695,E2 -22328.695} C_VEL
LIN {X 0,Y 185.729,Z 182.837,A -85,B 0,C 180,E1 -22333.124,E2 -22333.124} C_VEL
LIN {X 0,Y 185.69,Z 182.809,A -85,B 0,C 180,E1 -22337.626,E2 -22337.626} C_VEL
LIN {X 0,Y 185.597,Z 182.858,A -85,B 0,C 180,E1 -22342.252,E2 -22342.252} C_VEL
LIN {X 0,Y 185.563,Z 182.831,A -85,B 0,C 180,E1 -22347.033,E2 -22347.033} C_VEL
LIN {X 0,Y 185.58,Z 182.852,A -85,B 0,C 180,E1 -22349.494,E2 -22349.494} C_VEL
LIN {X 0,Y 185.501,Z 182.848,A -85,B 0,C 180,E1 -22354.633,E2 -22354.633} C_VEL
LIN {X 0,Y 185.509,Z 182.879,A -85,B 0,C 180,E1 -22357.314,E2 -22357.314} C_VEL
LIN {X 0,Y 185.493,Z 183.059,A -85,B 0,C 180,E1 -22360.429,E2 -22360.429} C_VEL
LIN {X 0,Y 186.144,Z 185.51,A -85,B 0,C 180,E1 -22362.503,E2 -22362.503} C_VEL
LIN {X 0,Y 187.502,Z 188.41,A -85,B 0,C 180,E1 -22363.287,E2 -22363.287} C_VEL
LIN {X 0,Y 189.844,Z 191.825,A -85,B 0,C 180,E1 -22364.209,E2 -22364.209} C_VEL
LIN {X 0,Y 197.704,Z 205.515,A -85,B 0,C 180,E1 -22367.155,E2 -22367.155} C_VEL
LIN {X 0,Y 204.044,Z 218.455,A -85,B 0,C 180,E1 -22369.363,E2 -22369.363} C_VEL
LIN {X 0,Y 210.112,Z 232.942,A -85,B 0,C 180,E1 -22371.381,E2 -22371.381} C_VEL
LIN {X 0,Y 210.881,Z 236.577,A -85,B 0,C 180,E1 -22371.701,E2 -22371.701} C_VEL
LIN {X 0,Y 212.673,Z 248.708,A -85,B 0,C 180,E1 -22372.585,E2 -22372.585} C_VEL
LIN {X 0,Y 210.51,Z 291.957,A -85,B 0,C 180,E1 -22374.002,E2 -22374.002} C_VEL
LIN {X 0,Y 209.43,Z 302.699,A -85,B 0,C 180,E1 -22374.56,E2 -22374.56} C_VEL
LIN {X 0,Y 207.776,Z 313.445,A -85,B 0,C 180,E1 -22375.342,E2 -22375.342} C_VEL
LIN {X 0,Y 205.468,Z 325.255,A -85,B 0,C 180,E1 -22376.527,E2 -22376.527} C_VEL
LIN {X 0,Y 202.741,Z 336.649,A -85,B 0,C 180,E1 -22378.087,E2 -22378.087} C_VEL
LIN {X 0,Y 199.737,Z 346.939,A -85,B 0,C 180,E1 -22379.907,E2 -22379.907} C_VEL
LIN {X 0,Y 197.024,Z 355.463,A -85,B 0,C 180,E1 -22381.795,E2 -22381.795} C_VEL
LIN {X 0,Y 194.55,Z 362.679,A -85,B 0,C 180,E1 -22383.735,E2 -22383.735} C_VEL
LIN {X 0,Y 192.332,Z 368.879,A -85,B 0,C 180,E1 -22385.727,E2 -22385.727} C_VEL
LIN {X 0,Y 190.065,Z 375.419,A -85,B 0,C 180,E1 -22388.299,E2 -22388.299} C_VEL
LIN {X 0,Y 188.321,Z 379.919,A -85,B 0,C 180,E1 -22390.375,E2 -22390.375} C_VEL
LIN {X 0,Y 186.187,Z 385.41,A -85,B 0,C 180,E1 -22393.555,E2 -22393.555} C_VEL
LIN {X 0,Y 184.682,Z 389.738,A -85,B 0,C 180,E1 -22396.802,E2 -22396.802} C_VEL
LIN {X 0,Y 184.033,Z 391.9,A -85,B 0,C 180,E1 -22398.79,E2 -22398.79} C_VEL
LIN {X 0,Y 182.946,Z 393.55,A -85,B 0,C 180,E1 -22400.529,E2 -22400.529} C_VEL
LIN {X 0,Y 179.666,Z 395.493,A -85,B 0,C 180,E1 -22403.422,E2 -22403.422} C_VEL
LIN {X 0,Y 177.102,Z 396.404,A -85,B 0,C 180,E1 -22405.838,E2 -22405.838} C_VEL
LIN {X 0,Y 176.045,Z 396.781,A -85,B 0,C 180,E1 -22407.739,E2 -22407.739} C_VEL
LIN {X 0,Y 175.968,Z 396.818,A -85,B 0,C 180,E1 -22408.385,E2 -22408.385} C_VEL
LIN {X 0,Y 176.058,Z 396.93,A -85,B 0,C 180,E1 -22410,E2 -22410} C_VEL
LIN {X 0,Y 175.95,Z 396.578,A -85,B 0,C 180,E1 -22413.037,E2 -22413.037} C_VEL
LIN {X 0,Y 176.092,Z 395.112,A -85,B 0,C 180,E1 -22416.877,E2 -22416.877} C_VEL
LIN {X 0,Y 176.424,Z 393.72,A -85,B 0,C 180,E1 -22419.169,E2 -22419.169} C_VEL
LIN {X 0,Y 177.339,Z 390.765,A -85,B 0,C 180,E1 -22422.589,E2 -22422.589} C_VEL
LIN {X 0,Y 178.705,Z 386.771,A -85,B 0,C 180,E1 -22425.979,E2 -22425.979} C_VEL
LIN {X 0,Y 180.839,Z 381.643,A -85,B 0,C 180,E1 -22429.289,E2 -22429.289} C_VEL
LIN {X 0,Y 182.972,Z 376.382,A -85,B 0,C 180,E1 -22431.993,E2 -22431.993} C_VEL
LIN {X 0,Y 185.399,Z 370.064,A -85,B 0,C 180,E1 -22434.644,E2 -22434.644} C_VEL
LIN {X 0,Y 187.574,Z 364.113,A -85,B 0,C 180,E1 -22436.719,E2 -22436.719} C_VEL
LIN {X 0,Y 190.105,Z 357.189,A -85,B 0,C 180,E1 -22438.724,E2 -22438.724} C_VEL
LIN {X 0,Y 192.874,Z 349.014,A -85,B 0,C 180,E1 -22440.673,E2 -22440.673} C_VEL
LIN {X 0,Y 195.505,Z 340.508,A -85,B 0,C 180,E1 -22442.325,E2 -22442.325} C_VEL
LIN {X 0,Y 197.94,Z 331.798,A -85,B 0,C 180,E1 -22443.695,E2 -22443.695} C_VEL
LIN {X 0,Y 200.195,Z 322.043,A -85,B 0,C 180,E1 -22444.936,E2 -22444.936} C_VEL
LIN {X 0,Y 202.16,Z 311.965,A -85,B 0,C 180,E1 -22445.919,E2 -22445.919} C_VEL
LIN {X 0,Y 203.689,Z 302.276,A -85,B 0,C 180,E1 -22446.618,E2 -22446.618} C_VEL
LIN {X 0,Y 204.721,Z 291.984,A -85,B 0,C 180,E1 -22447.165,E2 -22447.165} C_VEL
LIN {X 0,Y 207.014,Z 249.264,A -85,B 0,C 180,E1 -22448.591,E2 -22448.591} C_VEL
LIN {X 0,Y 204.934,Z 236.111,A -85,B 0,C 180,E1 -22449.636,E2 -22449.636} C_VEL
LIN {X 0,Y 199.471,Z 222.834,A -85,B 0,C 180,E1 -22451.56,E2 -22451.56} C_VEL
LIN {X 0,Y 193.179,Z 209.716,A -85,B 0,C 180,E1 -22453.882,E2 -22453.882} C_VEL
LIN {X 0,Y 185.418,Z 195.937,A -85,B 0,C 180,E1 -22456.978,E2 -22456.978} C_VEL
LIN {X 0,Y 182.556,Z 191.43,A -85,B 0,C 180,E1 -22458.202,E2 -22458.202} C_VEL
LIN {X 0,Y 179.296,Z 186.502,A -85,B 0,C 180,E1 -22459.7,E2 -22459.7} C_VEL
LIN {X 0,Y 178.688,Z 185.036,A -85,B 0,C 180,E1 -22460.271,E2 -22460.271} C_VEL
LIN {X 0,Y 178.411,Z 183.795,A -85,B 0,C 180,E1 -22461.549,E2 -22461.549} C_VEL
LIN {X 0,Y 178.488,Z 183.722,A -85,B 0,C 180,E1 -22466.546,E2 -22466.546} C_VEL
LIN {X 0,Y 178.524,Z 183.739,A -85,B 0,C 180,E1 -22470.005,E2 -22470.005} C_VEL
LIN {X 0,Y 178.525,Z 183.717,A -85,B 0,C 180,E1 -22474.881,E2 -22474.881} C_VEL
LIN {X 0,Y 178.623,Z 183.686,A -85,B 0,C 180,E1 -22480.783,E2 -22480.783} C_VEL
LIN {X 0,Y 178.658,Z 183.724,A -85,B 0,C 180,E1 -22486.347,E2 -22486.347} C_VEL
LIN {X 0,Y 178.911,Z 183.646,A -85,B 0,C 180,E1 -22490.959,E2 -22490.959} C_VEL
LIN {X 0,Y 178.868,Z 183.705,A -85,B 0,C 180,E1 -22495.492,E2 -22495.492} C_VEL
LIN {X 0,Y 179.366,Z 183.587,A -85,B 0,C 180,E1 -22499.999,E2 -22499.999} C_VEL
LIN {X 0,Y 178.873,Z 183.702,A -85,B 0,C 180,E1 -22504.506,E2 -22504.506} C_VEL
LIN {X 0,Y 178.937,Z 183.645,A -85,B 0,C 180,E1 -22509.038,E2 -22509.038} C_VEL
LIN {X 0,Y 178.685,Z 183.72,A -85,B 0,C 180,E1 -22513.649,E2 -22513.649} C_VEL
LIN {X 0,Y 178.648,Z 183.686,A -85,B 0,C 180,E1 -22518.343,E2 -22518.343} C_VEL
LIN {X 0,Y 178.51,Z 183.75,A -85,B 0,C 180,E1 -22523.184,E2 -22523.184} C_VEL
LIN {X 0,Y 178.484,Z 183.716,A -85,B 0,C 180,E1 -22528.196,E2 -22528.196} C_VEL
LIN {X 0,Y 178.498,Z 183.751,A -85,B 0,C 180,E1 -22530.786,E2 -22530.786} C_VEL
LIN {X 0,Y 178.488,Z 183.721,A -85,B 0,C 180,E1 -22534.222,E2 -22534.222} C_VEL
LIN {X 0,Y 178.473,Z 183.905,A -85,B 0,C 180,E1 -22539.783,E2 -22539.783} C_VEL
LIN {X 0,Y 178.709,Z 184.982,A -85,B 0,C 180,E1 -22540.363,E2 -22540.363} C_VEL
LIN {X 0,Y 180.32,Z 187.76,A -85,B 0,C 180,E1 -22541.164,E2 -22541.164} C_VEL
LIN {X 0,Y 181.865,Z 189.168,A -85,B 0,C 180,E1 -22541.804,E2 -22541.804} C_VEL
LIN {X 0,Y 183.918,Z 192.491,A -85,B 0,C 180,E1 -22542.707,E2 -22542.707} C_VEL
LIN {X 0,Y 185.408,Z 194.328,A -85,B 0,C 180,E1 -22543.309,E2 -22543.309} C_VEL
LIN {X 0,Y 193.246,Z 205.893,A -85,B 0,C 180,E1 -22546.324,E2 -22546.324} C_VEL
LIN {X 0,Y 200.425,Z 217.975,A -85,B 0,C 180,E1 -22548.833,E2 -22548.833} C_VEL
LIN {X 0,Y 207.843,Z 232.595,A -85,B 0,C 180,E1 -22551.248,E2 -22551.248} C_VEL
LIN {X 0,Y 216.397,Z 250.642,A -85,B 0,C 180,E1 -22553.788,E2 -22553.788} C_VEL
LIN {X 0,Y 225.071,Z 264.86,A -85,B 0,C 180,E1 -22555.939,E2 -22555.939} C_VEL
LIN {X 0,Y 233.128,Z 275.96,A -85,B 0,C 180,E1 -22557.675,E2 -22557.675} C_VEL
LIN {X 0,Y 243.301,Z 288.064,A -85,B 0,C 180,E1 -22559.752,E2 -22559.752} C_VEL
LIN {X 0,Y 254.498,Z 300.064,A -85,B 0,C 180,E1 -22562.088,E2 -22562.088} C_VEL
LIN {X 0,Y 266.63,Z 311.172,A -85,B 0,C 180,E1 -22564.524,E2 -22564.524} C_VEL
LIN {X 0,Y 279.939,Z 321.769,A -85,B 0,C 180,E1 -22567.06,E2 -22567.06} C_VEL
LIN {X 0,Y 292.765,Z 331.192,A -85,B 0,C 180,E1 -22569.423,E2 -22569.423} C_VEL
LIN {X 0,Y 300.157,Z 336.645,A -85,B 0,C 180,E1 -22570.865,E2 -22570.865} C_VEL
LIN {X 0,Y 307.414,Z 341.764,A -85,B 0,C 180,E1 -22572.426,E2 -22572.426} C_VEL
LIN {X 0,Y 311.624,Z 344.681,A -85,B 0,C 180,E1 -22573.429,E2 -22573.429} C_VEL
LIN {X 0,Y 316.749,Z 348.423,A -85,B 0,C 180,E1 -22574.829,E2 -22574.829} C_VEL
LIN {X 0,Y 322.008,Z 351.791,A -85,B 0,C 180,E1 -22576.35,E2 -22576.35} C_VEL
LIN {X 0,Y 327.083,Z 354.928,A -85,B 0,C 180,E1 -22578.013,E2 -22578.013} C_VEL
LIN {X 0,Y 331.131,Z 357.816,A -85,B 0,C 180,E1 -22579.67,E2 -22579.67} C_VEL
LIN {X 0,Y 335.064,Z 360.387,A -85,B 0,C 180,E1 -22581.557,E2 -22581.557} C_VEL
LIN {X 0,Y 337.428,Z 361.662,A -85,B 0,C 180,E1 -22582.821,E2 -22582.821} C_VEL
LIN {X 0,Y 339.423,Z 362.651,A -85,B 0,C 180,E1 -22584.058,E2 -22584.058} C_VEL
LIN {X 0,Y 341.104,Z 363.375,A -85,B 0,C 180,E1 -22585.273,E2 -22585.273} C_VEL
LIN {X 0,Y 342.448,Z 363.861,A -85,B 0,C 180,E1 -22586.47,E2 -22586.47} C_VEL
LIN {X 0,Y 343.323,Z 364.225,A -85,B 0,C 180,E1 -22587.654,E2 -22587.654} C_VEL
LIN {X 0,Y 343.774,Z 364.49,A -85,B 0,C 180,E1 -22588.829,E2 -22588.829} C_VEL
LIN {X 0,Y 344.061,Z 364.461,A -85,B 0,C 180,E1 -22590,E2 -22590} C_VEL
LIN {X 0,Y 343.793,Z 364.46,A -85,B 0,C 180,E1 -22591.171,E2 -22591.171} C_VEL
LIN {X 0,Y 343.323,Z 364.202,A -85,B 0,C 180,E1 -22592.346,E2 -22592.346} C_VEL
LIN {X 0,Y 342.444,Z 363.834,A -85,B 0,C 180,E1 -22593.53,E2 -22593.53} C_VEL
LIN {X 0,Y 341.092,Z 363.349,A -85,B 0,C 180,E1 -22594.727,E2 -22594.727} C_VEL
LIN {X 0,Y 339.228,Z 362.563,A -85,B 0,C 180,E1 -22596.05,E2 -22596.05} C_VEL
LIN {X 0,Y 337.399,Z 361.658,A -85,B 0,C 180,E1 -22597.18,E2 -22597.18} C_VEL
LIN {X 0,Y 334.292,Z 359.883,A -85,B 0,C 180,E1 -22598.851,E2 -22598.851} C_VEL
LIN {X 0,Y 331.127,Z 357.83,A -85,B 0,C 180,E1 -22600.326,E2 -22600.326} C_VEL
LIN {X 0,Y 325.772,Z 354.065,A -85,B 0,C 180,E1 -22602.458,E2 -22602.458} C_VEL
LIN {X 0,Y 321.081,Z 351.216,A -85,B 0,C 180,E1 -22603.932,E2 -22603.932} C_VEL
LIN {X 0,Y 314.189,Z 346.639,A -85,B 0,C 180,E1 -22605.88,E2 -22605.88} C_VEL
LIN {X 0,Y 307.407,Z 341.793,A -85,B 0,C 180,E1 -22607.574,E2 -22607.574} C_VEL
LIN {X 0,Y 300.157,Z 336.676,A -85,B 0,C 180,E1 -22609.135,E2 -22609.135} C_VEL
LIN {X 0,Y 292.769,Z 331.175,A -85,B 0,C 180,E1 -22610.579,E2 -22610.579} C_VEL
LIN {X 0,Y 278.073,Z 320.368,A -85,B 0,C 180,E1 -22613.287,E2 -22613.287} C_VEL
LIN {X 0,Y 265.28,Z 309.985,A -85,B 0,C 180,E1 -22615.745,E2 -22615.745} C_VEL
LIN {X 0,Y 253.577,Z 299.097,A -85,B 0,C 180,E1 -22618.109,E2 -22618.109} C_VEL
LIN {X 0,Y 242.63,Z 287.287,A -85,B 0,C 180,E1 -22620.387,E2 -22620.387} C_VEL
LIN {X 0,Y 232.649,Z 275.366,A -85,B 0,C 180,E1 -22622.422,E2 -22622.422} C_VEL
LIN {X 0,Y 222.435,Z 260.875,A -85,B 0,C 180,E1 -22624.678,E2 -22624.678} C_VEL
LIN {X 0,Y 214.582,Z 247.114,A -85,B 0,C 180,E1 -22626.715,E2 -22626.715} C_VEL
LIN {X 0,Y 205.198,Z 227.218,A -85,B 0,C 180,E1 -22629.591,E2 -22629.591} C_VEL
LIN {X 0,Y 198.366,Z 214.326,A -85,B 0,C 180,E1 -22631.867,E2 -22631.867} C_VEL
LIN {X 0,Y 191.856,Z 203.813,A -85,B 0,C 180,E1 -22634.183,E2 -22634.183} C_VEL
LIN {X 0,Y 187.084,Z 196.842,A -85,B 0,C 180,E1 -22636.009,E2 -22636.009} C_VEL
LIN {X 0,Y 184.6,Z 193.176,A -85,B 0,C 180,E1 -22637.024,E2 -22637.024} C_VEL
LIN {X 0,Y 182.354,Z 190.224,A -85,B 0,C 180,E1 -22637.962,E2 -22637.962} C_VEL
LIN {X 0,Y 181.603,Z 188.845,A -85,B 0,C 180,E1 -22638.308,E2 -22638.308} C_VEL
LIN {X 0,Y 179.44,Z 186.59,A -85,B 0,C 180,E1 -22639.231,E2 -22639.231} C_VEL
LIN {X 0,Y 178.552,Z 184.323,A -85,B 0,C 180,E1 -22639.871,E2 -22639.871} C_VEL
LIN {X 0,Y 178.435,Z 183.787,A -85,B 0,C 180,E1 -22640.573,E2 -22640.573} C_VEL
LIN {X 0,Y 178.488,Z 183.721,A -85,B 0,C 180,E1 -22645.778,E2 -22645.778} C_VEL
LIN {X 0,Y 178.52,Z 183.734,A -85,B 0,C 180,E1 -22650.007,E2 -22650.007} C_VEL
LIN {X 0,Y 178.532,Z 183.723,A -85,B 0,C 180,E1 -22654.877,E2 -22654.877} C_VEL
LIN {X 0,Y 178.621,Z 183.688,A -85,B 0,C 180,E1 -22660.785,E2 -22660.785} C_VEL
LIN {X 0,Y 178.664,Z 183.714,A -85,B 0,C 180,E1 -22664.018,E2 -22664.018} C_VEL
LIN {X 0,Y 178.86,Z 183.656,A -85,B 0,C 180,E1 -22669.211,E2 -22669.211} C_VEL
LIN {X 0,Y 178.924,Z 183.677,A -85,B 0,C 180,E1 -22673.234,E2 -22673.234} C_VEL
LIN {X 0,Y 179.153,Z 183.629,A -85,B 0,C 180,E1 -22677.753,E2 -22677.753} C_VEL
LIN {X 0,Y 179.366,Z 183.587,A -85,B 0,C 180,E1 -22680.001,E2 -22680.001} C_VEL
LIN {X 0,Y 178.868,Z 183.705,A -85,B 0,C 180,E1 -22684.508,E2 -22684.508} C_VEL
LIN {X 0,Y 178.911,Z 183.646,A -85,B 0,C 180,E1 -22689.041,E2 -22689.041} C_VEL
LIN {X 0,Y 178.658,Z 183.724,A -85,B 0,C 180,E1 -22693.653,E2 -22693.653} C_VEL
LIN {X 0,Y 178.623,Z 183.686,A -85,B 0,C 180,E1 -22699.217,E2 -22699.217} C_VEL
LIN {X 0,Y 178.525,Z 183.717,A -85,B 0,C 180,E1 -22705.119,E2 -22705.119} C_VEL
LIN {X 0,Y 178.502,Z 183.751,A -85,B 0,C 180,E1 -22710.788,E2 -22710.788} C_VEL
LIN {X 0,Y 178.486,Z 183.72,A -85,B 0,C 180,E1 -22714.221,E2 -22714.221} C_VEL
LIN {X 0,Y 178.425,Z 183.947,A -85,B 0,C 180,E1 -22718.757,E2 -22718.757} C_VEL
LIN {X 0,Y 178.918,Z 185.599,A -85,B 0,C 180,E1 -22720.034,E2 -22720.034} C_VEL
LIN {X 0,Y 181.26,Z 189.632,A -85,B 0,C 180,E1 -22721.236,E2 -22721.236} C_VEL
LIN {X 0,Y 182.937,Z 192.091,A -85,B 0,C 180,E1 -22721.969,E2 -22721.969} C_VEL
LIN {X 0,Y 186.461,Z 197.891,A -85,B 0,C 180,E1 -22723.469,E2 -22723.469} C_VEL
LIN {X 0,Y 193.334,Z 210.035,A -85,B 0,C 180,E1 -22726.178,E2 -22726.178} C_VEL
LIN {X 0,Y 199.378,Z 222.63,A -85,B 0,C 180,E1 -22728.407,E2 -22728.407} C_VEL
LIN {X 0,Y 205.131,Z 236.698,A -85,B 0,C 180,E1 -22730.436,E2 -22730.436} C_VEL
LIN {X 0,Y 207.031,Z 249.877,A -85,B 0,C 180,E1 -22731.439,E2 -22731.439} C_VEL
LIN {X 0,Y 204.788,Z 292.118,A -85,B 0,C 180,E1 -22732.851,E2 -22732.851} C_VEL
LIN {X 0,Y 203.55,Z 303.521,A -85,B 0,C 180,E1 -22733.462,E2 -22733.462} C_VEL
LIN {X 0,Y 201.517,Z 315.826,A -85,B 0,C 180,E1 -22734.41,E2 -22734.41} C_VEL
LIN {X 0,Y 198.717,Z 328.534,A -85,B 0,C 180,E1 -22735.844,E2 -22735.844} C_VEL
LIN {X 0,Y 196.35,Z 337.808,A -85,B 0,C 180,E1 -22737.223,E2 -22737.223} C_VEL
LIN {X 0,Y 193.617,Z 346.747,A -85,B 0,C 180,E1 -22738.852,E2 -22738.852} C_VEL
LIN {X 0,Y 190.784,Z 355.271,A -85,B 0,C 180,E1 -22740.785,E2 -22740.785} C_VEL
LIN {X 0,Y 188.175,Z 362.486,A -85,B 0,C 180,E1 -22742.773,E2 -22742.773} C_VEL
LIN {X 0,Y 185.855,Z 368.686,A -85,B 0,C 180,E1 -22744.824,E2 -22744.824} C_VEL
LIN {X 0,Y 183.454,Z 375.227,A -85,B 0,C 180,E1 -22747.475,E2 -22747.475} C_VEL
LIN {X 0,Y 181.596,Z 379.726,A -85,B 0,C 180,E1 -22749.616,E2 -22749.616} C_VEL
LIN {X 0,Y 179.366,Z 385.218,A -85,B 0,C 180,E1 -22752.911,E2 -22752.911} C_VEL
LIN {X 0,Y 177.745,Z 389.546,A -85,B 0,C 180,E1 -22756.277,E2 -22756.277} C_VEL
LIN {X 0,Y 176.977,Z 391.942,A -85,B 0,C 180,E1 -22758.58,E2 -22758.58} C_VEL
LIN {X 0,Y 176.46,Z 393.721,A -85,B 0,C 180,E1 -22760.833,E2 -22760.833} C_VEL
LIN {X 0,Y 176.01,Z 396.178,A -85,B 0,C 180,E1 -22765.42,E2 -22765.42} C_VEL
LIN {X 0,Y 175.968,Z 396.818,A -85,B 0,C 180,E1 -22768.385,E2 -22768.385} C_VEL
LIN {X 0,Y 175.294,Z 396.927,A -85,B 0,C 180,E1 -22770.295,E2 -22770.295} C_VEL
LIN {X 0,Y 173.682,Z 396.747,A -85,B 0,C 180,E1 -22772.173,E2 -22772.173} C_VEL
LIN {X 0,Y 170.032,Z 395.526,A -85,B 0,C 180,E1 -22775.971,E2 -22775.971} C_VEL
LIN {X 0,Y 169.174,Z 394.366,A -85,B 0,C 180,E1 -22778.277,E2 -22778.277} C_VEL
LIN {X 0,Y 169.206,Z 394.079,A -85,B 0,C 180,E1 -22778.609,E2 -22778.609} C_VEL
LIN {X 0,Y 170.012,Z 391.725,A -85,B 0,C 180,E1 -22781.928,E2 -22781.928} C_VEL
LIN {X 0,Y 171.29,Z 388.11,A -85,B 0,C 180,E1 -22785.467,E2 -22785.467} C_VEL
LIN {X 0,Y 173.317,Z 383.366,A -85,B 0,C 180,E1 -22788.929,E2 -22788.929} C_VEL
